LIN {X 0,Y 658.001,Z 1135.753,A -85,B 0,C 180,E1 30891.202,E2 30891.202} C_VEL
LIN {X 0,Y 657.305,Z 1150.031,A -85,B 0,C 180,E1 30888.997,E2 30888.997} C_VEL
LIN {X 0,Y 656.752,Z 1162.678,A -85,B 0,C 180,E1 30886.723,E2 30886.723} C_VEL
LIN {X 0,Y 656.451,Z 1171.896,A -85,B 0,C 180,E1 30884.826,E2 30884.826} C_VEL
LIN {X 0,Y 656.232,Z 1179.871,A -85,B 0,C 180,E1 30882.943,E2 30882.943} C_VEL
LIN {X 0,Y 656.05,Z 1187.892,A -85,B 0,C 180,E1 30880.716,E2 30880.716} C_VEL
LIN {X 0,Y 655.97,Z 1194.694,A -85,B 0,C 180,E1 30878.326,E2 30878.326} C_VEL
LIN {X 0,Y 655.929,Z 1199.41,A -85,B 0,C 180,E1 30876.125,E2 30876.125} C_VEL
LIN {X 0,Y 655.91,Z 1202.789,A -85,B 0,C 180,E1 30873.846,E2 30873.846} C_VEL
LIN {X 0,Y 655.911,Z 1204.624,A -85,B 0,C 180,E1 30871.485,E2 30871.485} C_VEL
LIN {X 0,Y 655.893,Z 1204.849,A -85,B 0,C 180,E1 30869.389,E2 30869.389} C_VEL
LIN {X 0,Y 655.908,Z 1203.947,A -85,B 0,C 180,E1 30867.379,E2 30867.379} C_VEL
LIN {X 0,Y 655.919,Z 1201.428,A -85,B 0,C 180,E1 30865.103,E2 30865.103} C_VEL
LIN {X 0,Y 655.949,Z 1197.152,A -85,B 0,C 180,E1 30862.732,E2 30862.732} C_VEL
LIN {X 0,Y 656.009,Z 1191.376,A -85,B 0,C 180,E1 30860.437,E2 30860.437} C_VEL
LIN {X 0,Y 656.126,Z 1184.279,A -85,B 0,C 180,E1 30858.217,E2 30858.217} C_VEL
LIN {X 0,Y 656.39,Z 1174.089,A -85,B 0,C 180,E1 30855.658,E2 30855.658} C_VEL
LIN {X 0,Y 656.694,Z 1164.274,A -85,B 0,C 180,E1 30853.587,E2 30853.587} C_VEL
LIN {X 0,Y 657.112,Z 1154.137,A -85,B 0,C 180,E1 30851.716,E2 30851.716} C_VEL
LIN {X 0,Y 657.764,Z 1140.78,A -85,B 0,C 180,E1 30849.536,E2 30849.536} C_VEL
LIN {X 0,Y 658.6,Z 1125.104,A -85,B 0,C 180,E1 30847.318,E2 30847.318} C_VEL
LIN {X 0,Y 659.475,Z 1110.399,A -85,B 0,C 180,E1 30845.467,E2 30845.467} C_VEL
LIN {X 0,Y 660.73,Z 1092.314,A -85,B 0,C 180,E1 30843.428,E2 30843.428} C_VEL
LIN {X 0,Y 662,Z 1073.819,A -85,B 0,C 180,E1 30841.591,E2 30841.591} C_VEL
LIN {X 0,Y 663.289,Z 1056.842,A -85,B 0,C 180,E1 30840.069,E2 30840.069} C_VEL
LIN {X 0,Y 664.962,Z 1035.53,A -85,B 0,C 180,E1 30838.348,E2 30838.348} C_VEL
LIN {X 0,Y 666.618,Z 1013.004,A -85,B 0,C 180,E1 30836.756,E2 30836.756} C_VEL
LIN {X 0,Y 668.131,Z 993.022,A -85,B 0,C 180,E1 30835.499,E2 30835.499} C_VEL
LIN {X 0,Y 669.972,Z 968.967,A -85,B 0,C 180,E1 30834.161,E2 30834.161} C_VEL
LIN {X 0,Y 671.656,Z 944.001,A -85,B 0,C 180,E1 30832.976,E2 30832.976} C_VEL
LIN {X 0,Y 672.975,Z 923.055,A -85,B 0,C 180,E1 30832.114,E2 30832.114} C_VEL
LIN {X 0,Y 674.098,Z 902.837,A -85,B 0,C 180,E1 30831.392,E2 30831.392} C_VEL
LIN {X 0,Y 675.312,Z 879.657,A -85,B 0,C 180,E1 30830.692,E2 30830.692} C_VEL
LIN {X 0,Y 676.519,Z 851.801,A -85,B 0,C 180,E1 30830.029,E2 30830.029} C_VEL
LIN {X 0,Y 677.299,Z 826.241,A -85,B 0,C 180,E1 30829.585,E2 30829.585} C_VEL
LIN {X 0,Y 680.373,Z 611.931,A -85,B 0,C 180,E1 30826.813,E2 30826.813} C_VEL
LIN {X 0,Y 683.542,Z 400.047,A -85,B 0,C 180,E1 30824.005,E2 30824.005} C_VEL
LIN {X 0,Y 683.78,Z 375.573,A -85,B 0,C 180,E1 30823.663,E2 30823.663} C_VEL
LIN {X 0,Y 678.293,Z 349.765,A -85,B 0,C 180,E1 30822.77,E2 30822.77} C_VEL
LIN {X 0,Y 678.555,Z 340.602,A -85,B 0,C 180,E1 30822.168,E2 30822.168} C_VEL
LIN {X 0,Y 667.4,Z 318.931,A -85,B 0,C 180,E1 30819.66,E2 30819.66} C_VEL
LIN {X 0,Y 660.624,Z 305.776,A -85,B 0,C 180,E1 30818.026,E2 30818.026} C_VEL
LIN {X 0,Y 658.168,Z 301.139,A -85,B 0,C 180,E1 30817.422,E2 30817.422} C_VEL
LIN {X 0,Y 656.727,Z 297.652,A -85,B 0,C 180,E1 30816.96,E2 30816.96} C_VEL
LIN {X 0,Y 656.684,Z 297.427,A -85,B 0,C 180,E1 30813.974,E2 30813.974} C_VEL
LIN {X 0,Y 656.694,Z 297.401,A -85,B 0,C 180,E1 30810.974,E2 30810.974} C_VEL
LIN {X 0,Y 656.692,Z 297.415,A -85,B 0,C 180,E1 30807.967,E2 30807.967} C_VEL
LIN {X 0,Y 656.698,Z 297.426,A -85,B 0,C 180,E1 30804.946,E2 30804.946} C_VEL
LIN {X 0,Y 656.696,Z 297.397,A -85,B 0,C 180,E1 30801.903,E2 30801.903} C_VEL
LIN {X 0,Y 656.699,Z 297.431,A -85,B 0,C 180,E1 30798.832,E2 30798.832} C_VEL
LIN {X 0,Y 656.694,Z 297.39,A -85,B 0,C 180,E1 30795.725,E2 30795.725} C_VEL
LIN {X 0,Y 656.695,Z 297.429,A -85,B 0,C 180,E1 30792.665,E2 30792.665} C_VEL
LIN {X 0,Y 656.696,Z 297.389,A -85,B 0,C 180,E1 30789.553,E2 30789.553} C_VEL
LIN {X 0,Y 656.689,Z 297.431,A -85,B 0,C 180,E1 30786.47,E2 30786.47} C_VEL
LIN {X 0,Y 656.702,Z 297.422,A -85,B 0,C 180,E1 30783.404,E2 30783.404} C_VEL
LIN {X 0,Y 656.686,Z 297.43,A -85,B 0,C 180,E1 30780.349,E2 30780.349} C_VEL
LIN {X 0,Y 656.703,Z 297.416,A -85,B 0,C 180,E1 30777.295,E2 30777.295} C_VEL
LIN {X 0,Y 656.686,Z 297.423,A -85,B 0,C 180,E1 30774.232,E2 30774.232} C_VEL
LIN {X 0,Y 656.707,Z 297.424,A -85,B 0,C 180,E1 30771.154,E2 30771.154} C_VEL
LIN {X 0,Y 656.682,Z 297.428,A -85,B 0,C 180,E1 30768.049,E2 30768.049} C_VEL
LIN {X 0,Y 656.71,Z 297.424,A -85,B 0,C 180,E1 30764.999,E2 30764.999} C_VEL
LIN {X 0,Y 656.678,Z 297.432,A -85,B 0,C 180,E1 30761.903,E2 30761.903} C_VEL
LIN {X 0,Y 656.709,Z 297.42,A -85,B 0,C 180,E1 30758.847,E2 30758.847} C_VEL
LIN {X 0,Y 656.67,Z 297.403,A -85,B 0,C 180,E1 30755.725,E2 30755.725} C_VEL
LIN {X 0,Y 656.705,Z 297.417,A -85,B 0,C 180,E1 30752.722,E2 30752.722} C_VEL
LIN {X 0,Y 656.67,Z 297.407,A -85,B 0,C 180,E1 30749.634,E2 30749.634} C_VEL
LIN {X 0,Y 656.698,Z 297.42,A -85,B 0,C 180,E1 30746.656,E2 30746.656} C_VEL
LIN {X 0,Y 656.666,Z 297.4,A -85,B 0,C 180,E1 30743.509,E2 30743.509} C_VEL
LIN {X 0,Y 656.695,Z 297.428,A -85,B 0,C 180,E1 30740.528,E2 30740.528} C_VEL
LIN {X 0,Y 656.698,Z 297.428,A -85,B 0,C 180,E1 30740.497,E2 30740.497} C_VEL
LIN {X 0,Y 655.768,Z 297.543,A -85,B 0,C 180,E1 30739.825,E2 30739.825} C_VEL
LIN {X 0,Y 649.201,Z 298.332,A -85,B 0,C 180,E1 30737.893,E2 30737.893} C_VEL
LIN {X 0,Y 648.731,Z 298.392,A -85,B 0,C 180,E1 30737.451,E2 30737.451} C_VEL
LIN {X 0,Y 648.729,Z 298.404,A -85,B 0,C 180,E1 30734.595,E2 30734.595} C_VEL
LIN {X 0,Y 648.737,Z 298.422,A -85,B 0,C 180,E1 30731.357,E2 30731.357} C_VEL
LIN {X 0,Y 648.807,Z 298.65,A -85,B 0,C 180,E1 30729.906,E2 30729.906} C_VEL
LIN {X 0,Y 650.17,Z 302.073,A -85,B 0,C 180,E1 30729.429,E2 30729.429} C_VEL
LIN {X 0,Y 656.974,Z 316.09,A -85,B 0,C 180,E1 30727.538,E2 30727.538} C_VEL
LIN {X 0,Y 663.735,Z 330.81,A -85,B 0,C 180,E1 30725.66,E2 30725.66} C_VEL
LIN {X 0,Y 667.446,Z 339.825,A -85,B 0,C 180,E1 30724.594,E2 30724.594} C_VEL
LIN {X 0,Y 667.126,Z 347.451,A -85,B 0,C 180,E1 30724.054,E2 30724.054} C_VEL
LIN {X 0,Y 673.211,Z 374.417,A -85,B 0,C 180,E1 30723.133,E2 30723.133} C_VEL
LIN {X 0,Y 669.499,Z 604.5,A -85,B 0,C 180,E1 30720.151,E2 30720.151} C_VEL
LIN {X 0,Y 667.067,Z 780.533,A -85,B 0,C 180,E1 30717.931,E2 30717.931} C_VEL
LIN {X 0,Y 666.246,Z 807.391,A -85,B 0,C 180,E1 30717.446,E2 30717.446} C_VEL
LIN {X 0,Y 665.258,Z 830.021,A -85,B 0,C 180,E1 30716.891,E2 30716.891} C_VEL
LIN {X 0,Y 664.302,Z 849.337,A -85,B 0,C 180,E1 30716.312,E2 30716.312} C_VEL
LIN {X 0,Y 663.135,Z 870.21,A -85,B 0,C 180,E1 30715.571,E2 30715.571} C_VEL
LIN {X 0,Y 661.528,Z 895.398,A -85,B 0,C 180,E1 30714.506,E2 30714.506} C_VEL
LIN {X 0,Y 660.09,Z 916.05,A -85,B 0,C 180,E1 30713.476,E2 30713.476} C_VEL
LIN {X 0,Y 658.632,Z 936.675,A -85,B 0,C 180,E1 30712.304,E2 30712.304} C_VEL
LIN {X 0,Y 656.942,Z 959.384,A -85,B 0,C 180,E1 30710.817,E2 30710.817} C_VEL
LIN {X 0,Y 655.495,Z 978.127,A -85,B 0,C 180,E1 30709.422,E2 30709.422} C_VEL
LIN {X 0,Y 654.046,Z 998.172,A -85,B 0,C 180,E1 30707.743,E2 30707.743} C_VEL
LIN {X 0,Y 652.711,Z 1016.296,A -85,B 0,C 180,E1 30706.006,E2 30706.006} C_VEL
LIN {X 0,Y 651.571,Z 1033.024,A -85,B 0,C 180,E1 30704.213,E2 30704.213} C_VEL
LIN {X 0,Y 650.501,Z 1049.809,A -85,B 0,C 180,E1 30702.156,E2 30702.156} C_VEL
LIN {X 0,Y 649.761,Z 1063.29,A -85,B 0,C 180,E1 30700.282,E2 30700.282} C_VEL
LIN {X 0,Y 649.074,Z 1077.256,A -85,B 0,C 180,E1 30698.058,E2 30698.058} C_VEL
LIN {X 0,Y 648.632,Z 1087.822,A -85,B 0,C 180,E1 30696.106,E2 30696.106} C_VEL
LIN {X 0,Y 648.338,Z 1097.37,A -85,B 0,C 180,E1 30694.068,E2 30694.068} C_VEL
LIN {X 0,Y 648.105,Z 1106.283,A -85,B 0,C 180,E1 30691.768,E2 30691.768} C_VEL
LIN {X 0,Y 647.99,Z 1112.419,A -85,B 0,C 180,E1 30689.823,E2 30689.823} C_VEL
LIN {X 0,Y 647.948,Z 1117.134,A -85,B 0,C 180,E1 30687.966,E2 30687.966} C_VEL
LIN {X 0,Y 647.907,Z 1121.473,A -85,B 0,C 180,E1 30685.663,E2 30685.663} C_VEL
LIN {X 0,Y 647.912,Z 1123.863,A -85,B 0,C 180,E1 30683.532,E2 30683.532} C_VEL
LIN {X 0,Y 647.91,Z 1124.829,A -85,B 0,C 180,E1 30681.659,E2 30681.659} C_VEL
LIN {X 0,Y 647.904,Z 1124.662,A -85,B 0,C 180,E1 30679.598,E2 30679.598} C_VEL
LIN {X 0,Y 647.916,Z 1122.754,A -85,B 0,C 180,E1 30677.248,E2 30677.248} C_VEL
LIN {X 0,Y 647.915,Z 1119.922,A -85,B 0,C 180,E1 30675.34,E2 30675.34} C_VEL
LIN {X 0,Y 647.959,Z 1116.115,A -85,B 0,C 180,E1 30673.505,E2 30673.505} C_VEL
LIN {X 0,Y 648.043,Z 1110.121,A -85,B 0,C 180,E1 30671.281,E2 30671.281} C_VEL
LIN {X 0,Y 648.202,Z 1102.181,A -85,B 0,C 180,E1 30669.031,E2 30669.031} C_VEL
LIN {X 0,Y 648.411,Z 1094.625,A -85,B 0,C 180,E1 30667.229,E2 30667.229} C_VEL
LIN {X 0,Y 648.775,Z 1084.74,A -85,B 0,C 180,E1 30665.199,E2 30665.199} C_VEL
LIN {X 0,Y 649.31,Z 1072.034,A -85,B 0,C 180,E1 30662.982,E2 30662.982} C_VEL
LIN {X 0,Y 649.949,Z 1059.761,A -85,B 0,C 180,E1 30661.115,E2 30661.115} C_VEL
LIN {X 0,Y 650.876,Z 1043.982,A -85,B 0,C 180,E1 30659.006,E2 30659.006} C_VEL
LIN {X 0,Y 651.867,Z 1028.543,A -85,B 0,C 180,E1 30657.201,E2 30657.201} C_VEL
LIN {X 0,Y 653.028,Z 1011.944,A -85,B 0,C 180,E1 30655.464,E2 30655.464} C_VEL
LIN {X 0,Y 654.458,Z 992.162,A -85,B 0,C 180,E1 30653.646,E2 30653.646} C_VEL
LIN {X 0,Y 655.805,Z 974.433,A -85,B 0,C 180,E1 30652.201,E2 30652.201} C_VEL
LIN {X 0,Y 657.481,Z 952.02,A -85,B 0,C 180,E1 30650.585,E2 30650.585} C_VEL
LIN {X 0,Y 658.943,Z 932.021,A -85,B 0,C 180,E1 30649.33,E2 30649.33} C_VEL
LIN {X 0,Y 660.527,Z 910.49,A -85,B 0,C 180,E1 30648.14,E2 30648.14} C_VEL
LIN {X 0,Y 662.114,Z 886.692,A -85,B 0,C 180,E1 30647.015,E2 30647.015} C_VEL
LIN {X 0,Y 663.382,Z 865.65,A -85,B 0,C 180,E1 30646.167,E2 30646.167} C_VEL
LIN {X 0,Y 664.58,Z 844.003,A -85,B 0,C 180,E1 30645.425,E2 30645.425} C_VEL
LIN {X 0,Y 665.807,Z 817,A -85,B 0,C 180,E1 30644.682,E2 30644.682} C_VEL
LIN {X 0,Y 666.623,Z 794.883,A -85,B 0,C 180,E1 30644.217,E2 30644.217} C_VEL
LIN {X 0,Y 667.316,Z 769.851,A -85,B 0,C 180,E1 30643.828,E2 30643.828} C_VEL
LIN {X 0,Y 670.628,Z 527.96,A -85,B 0,C 180,E1 30640.783,E2 30640.783} C_VEL
LIN {X 0,Y 673.17,Z 373.299,A -85,B 0,C 180,E1 30638.744,E2 30638.744} C_VEL
LIN {X 0,Y 667.143,Z 346.712,A -85,B 0,C 180,E1 30637.807,E2 30637.807} C_VEL
LIN {X 0,Y 667.583,Z 340.05,A -85,B 0,C 180,E1 30637.317,E2 30637.317} C_VEL
LIN {X 0,Y 661.902,Z 326.465,A -85,B 0,C 180,E1 30635.669,E2 30635.669} C_VEL
LIN {X 0,Y 654.624,Z 310.93,A -85,B 0,C 180,E1 30633.568,E2 30633.568} C_VEL
LIN {X 0,Y 652.075,Z 305.952,A -85,B 0,C 180,E1 30632.831,E2 30632.831} C_VEL
LIN {X 0,Y 650.535,Z 302.539,A -85,B 0,C 180,E1 30632.336,E2 30632.336} C_VEL
LIN {X 0,Y 648.827,Z 298.862,A -85,B 0,C 180,E1 30631.767,E2 30631.767} C_VEL
LIN {X 0,Y 648.76,Z 298.417,A -85,B 0,C 180,E1 30631.201,E2 30631.201} C_VEL
LIN {X 0,Y 648.766,Z 298.416,A -85,B 0,C 180,E1 30628.039,E2 30628.039} C_VEL
LIN {X 0,Y 648.748,Z 298.402,A -85,B 0,C 180,E1 30624.883,E2 30624.883} C_VEL
LIN {X 0,Y 648.757,Z 298.39,A -85,B 0,C 180,E1 30621.805,E2 30621.805} C_VEL
LIN {X 0,Y 648.752,Z 298.418,A -85,B 0,C 180,E1 30618.698,E2 30618.698} C_VEL
LIN {X 0,Y 648.756,Z 298.407,A -85,B 0,C 180,E1 30615.582,E2 30615.582} C_VEL
LIN {X 0,Y 648.751,Z 298.392,A -85,B 0,C 180,E1 30612.552,E2 30612.552} C_VEL
LIN {X 0,Y 648.757,Z 298.42,A -85,B 0,C 180,E1 30609.474,E2 30609.474} C_VEL
LIN {X 0,Y 648.751,Z 298.388,A -85,B 0,C 180,E1 30606.371,E2 30606.371} C_VEL
LIN {X 0,Y 648.753,Z 298.409,A -85,B 0,C 180,E1 30603.269,E2 30603.269} C_VEL
LIN {X 0,Y 648.753,Z 298.403,A -85,B 0,C 180,E1 30600.177,E2 30600.177} C_VEL
LIN {X 0,Y 648.75,Z 298.395,A -85,B 0,C 180,E1 30597.085,E2 30597.085} C_VEL
LIN {X 0,Y 648.753,Z 298.412,A -85,B 0,C 180,E1 30593.984,E2 30593.984} C_VEL
LIN {X 0,Y 648.747,Z 298.387,A -85,B 0,C 180,E1 30590.955,E2 30590.955} C_VEL
LIN {X 0,Y 648.758,Z 298.416,A -85,B 0,C 180,E1 30587.901,E2 30587.901} C_VEL
LIN {X 0,Y 648.747,Z 298.393,A -85,B 0,C 180,E1 30584.81,E2 30584.81} C_VEL
LIN {X 0,Y 648.761,Z 298.412,A -85,B 0,C 180,E1 30581.768,E2 30581.768} C_VEL
LIN {X 0,Y 648.749,Z 298.414,A -85,B 0,C 180,E1 30578.67,E2 30578.67} C_VEL
LIN {X 0,Y 648.76,Z 298.387,A -85,B 0,C 180,E1 30575.603,E2 30575.603} C_VEL
LIN {X 0,Y 648.75,Z 298.408,A -85,B 0,C 180,E1 30572.559,E2 30572.559} C_VEL
LIN {X 0,Y 648.764,Z 298.417,A -85,B 0,C 180,E1 30569.429,E2 30569.429} C_VEL
LIN {X 0,Y 648.746,Z 298.416,A -85,B 0,C 180,E1 30566.331,E2 30566.331} C_VEL
LIN {X 0,Y 648.783,Z 298.677,A -85,B 0,C 180,E1 30563.835,E2 30563.835} C_VEL
LIN {X 0,Y 650.131,Z 301.988,A -85,B 0,C 180,E1 30563.363,E2 30563.363} C_VEL
LIN {X 0,Y 651.245,Z 303.643,A -85,B 0,C 180,E1 30563.107,E2 30563.107} C_VEL
LIN {X 0,Y 658.408,Z 317.778,A -85,B 0,C 180,E1 30561.267,E2 30561.267} C_VEL
LIN {X 0,Y 671.527,Z 343.462,A -85,B 0,C 180,E1 30558.241,E2 30558.241} C_VEL
LIN {X 0,Y 672.392,Z 345.474,A -85,B 0,C 180,E1 30558.031,E2 30558.031} C_VEL
LIN {X 0,Y 672.364,Z 350.69,A -85,B 0,C 180,E1 30557.728,E2 30557.728} C_VEL
LIN {X 0,Y 678.337,Z 378.966,A -85,B 0,C 180,E1 30556.77,E2 30556.77} C_VEL
LIN {X 0,Y 674.876,Z 590.194,A -85,B 0,C 180,E1 30553.941,E2 30553.941} C_VEL
LIN {X 0,Y 671.51,Z 814.244,A -85,B 0,C 180,E1 30551.028,E2 30551.028} C_VEL
LIN {X 0,Y 670.692,Z 842.215,A -85,B 0,C 180,E1 30550.596,E2 30550.596} C_VEL
LIN {X 0,Y 669.734,Z 865.671,A -85,B 0,C 180,E1 30550.102,E2 30550.102} C_VEL
LIN {X 0,Y 668.493,Z 890.858,A -85,B 0,C 180,E1 30549.428,E2 30549.428} C_VEL
LIN {X 0,Y 666.809,Z 918.654,A -85,B 0,C 180,E1 30548.487,E2 30548.487} C_VEL
LIN {X 0,Y 665.363,Z 939.924,A -85,B 0,C 180,E1 30547.63,E2 30547.63} C_VEL
LIN {X 0,Y 663.854,Z 960.721,A -85,B 0,C 180,E1 30546.669,E2 30546.669} C_VEL
LIN {X 0,Y 662.097,Z 983.908,A -85,B 0,C 180,E1 30545.443,E2 30545.443} C_VEL
LIN {X 0,Y 660.055,Z 1008.604,A -85,B 0,C 180,E1 30543.932,E2 30543.932} C_VEL
LIN {X 0,Y 658.449,Z 1027.581,A -85,B 0,C 180,E1 30542.62,E2 30542.62} C_VEL
LIN {X 0,Y 656.823,Z 1047.086,A -85,B 0,C 180,E1 30541.118,E2 30541.118} C_VEL
LIN {X 0,Y 654.983,Z 1069.757,A -85,B 0,C 180,E1 30539.141,E2 30539.141} C_VEL
LIN {X 0,Y 653.645,Z 1086.388,A -85,B 0,C 180,E1 30537.514,E2 30537.514} C_VEL
LIN {X 0,Y 652.369,Z 1103.305,A -85,B 0,C 180,E1 30535.679,E2 30535.679} C_VEL
LIN {X 0,Y 651.104,Z 1121.565,A -85,B 0,C 180,E1 30533.436,E2 30533.436} C_VEL
LIN {X 0,Y 650.245,Z 1135.429,A -85,B 0,C 180,E1 30531.515,E2 30531.515} C_VEL
LIN {X 0,Y 649.487,Z 1149.549,A -85,B 0,C 180,E1 30529.313,E2 30529.313} C_VEL
LIN {X 0,Y 648.874,Z 1162.214,A -85,B 0,C 180,E1 30527.024,E2 30527.024} C_VEL
LIN {X 0,Y 648.513,Z 1171.487,A -85,B 0,C 180,E1 30525.103,E2 30525.103} C_VEL
LIN {X 0,Y 648.28,Z 1179.515,A -85,B 0,C 180,E1 30523.195,E2 30523.195} C_VEL
LIN {X 0,Y 648.084,Z 1187.034,A -85,B 0,C 180,E1 30521.112,E2 30521.112} C_VEL
LIN {X 0,Y 647.987,Z 1193.816,A -85,B 0,C 180,E1 30518.787,E2 30518.787} C_VEL
LIN {X 0,Y 647.935,Z 1199.101,A -85,B 0,C 180,E1 30516.372,E2 30516.372} C_VEL
LIN {X 0,Y 647.918,Z 1202.476,A -85,B 0,C 180,E1 30514.159,E2 30514.159} C_VEL
LIN {X 0,Y 647.908,Z 1204.549,A -85,B 0,C 180,E1 30511.769,E2 30511.769} C_VEL
LIN {X 0,Y 647.892,Z 1204.872,A -85,B 0,C 180,E1 30509.47,E2 30509.47} C_VEL
LIN {X 0,Y 647.909,Z 1203.944,A -85,B 0,C 180,E1 30507.347,E2 30507.347} C_VEL
LIN {X 0,Y 647.922,Z 1201.428,A -85,B 0,C 180,E1 30505.043,E2 30505.043} C_VEL
LIN {X 0,Y 647.951,Z 1197.152,A -85,B 0,C 180,E1 30502.642,E2 30502.642} C_VEL
LIN {X 0,Y 648.018,Z 1191.373,A -85,B 0,C 180,E1 30500.318,E2 30500.318} C_VEL
LIN {X 0,Y 648.146,Z 1184.279,A -85,B 0,C 180,E1 30498.07,E2 30498.07} C_VEL
LIN {X 0,Y 648.439,Z 1174.338,A -85,B 0,C 180,E1 30495.535,E2 30495.535} C_VEL
LIN {X 0,Y 648.771,Z 1164.544,A -85,B 0,C 180,E1 30493.434,E2 30493.434} C_VEL
LIN {X 0,Y 649.238,Z 1154.237,A -85,B 0,C 180,E1 30491.503,E2 30491.503} C_VEL
LIN {X 0,Y 649.924,Z 1141.364,A -85,B 0,C 180,E1 30489.372,E2 30489.372} C_VEL
LIN {X 0,Y 650.838,Z 1125.803,A -85,B 0,C 180,E1 30487.128,E2 30487.128} C_VEL
LIN {X 0,Y 651.804,Z 1111.152,A -85,B 0,C 180,E1 30485.252,E2 30485.252} C_VEL
LIN {X 0,Y 653.113,Z 1093.727,A -85,B 0,C 180,E1 30483.251,E2 30483.251} C_VEL
LIN {X 0,Y 654.547,Z 1074.832,A -85,B 0,C 180,E1 30481.337,E2 30481.337} C_VEL
LIN {X 0,Y 655.937,Z 1057.951,A -85,B 0,C 180,E1 30479.8,E2 30479.8} C_VEL
LIN {X 0,Y 657.511,Z 1039.194,A -85,B 0,C 180,E1 30478.254,E2 30478.254} C_VEL
LIN {X 0,Y 659.487,Z 1015.132,A -85,B 0,C 180,E1 30476.501,E2 30476.501} C_VEL
LIN {X 0,Y 661.142,Z 994.951,A -85,B 0,C 180,E1 30475.207,E2 30475.207} C_VEL
LIN {X 0,Y 662.831,Z 974.061,A -85,B 0,C 180,E1 30474.017,E2 30474.017} C_VEL
LIN {X 0,Y 664.822,Z 948.476,A -85,B 0,C 180,E1 30472.747,E2 30472.747} C_VEL
LIN {X 0,Y 666.407,Z 925.174,A -85,B 0,C 180,E1 30471.764,E2 30471.764} C_VEL
LIN {X 0,Y 667.661,Z 904.465,A -85,B 0,C 180,E1 30471.01,E2 30471.01} C_VEL
LIN {X 0,Y 668.911,Z 882.309,A -85,B 0,C 180,E1 30470.327,E2 30470.327} C_VEL
LIN {X 0,Y 670.161,Z 856.683,A -85,B 0,C 180,E1 30469.689,E2 30469.689} C_VEL
LIN {X 0,Y 671.132,Z 829.115,A -85,B 0,C 180,E1 30469.183,E2 30469.183} C_VEL
LIN {X 0,Y 672.99,Z 712.974,A -85,B 0,C 180,E1 30467.665,E2 30467.665} C_VEL
LIN {X 0,Y 676.471,Z 490.787,A -85,B 0,C 180,E1 30464.739,E2 30464.739} C_VEL
LIN {X 0,Y 678.217,Z 377.64,A -85,B 0,C 180,E1 30463.199,E2 30463.199} C_VEL
LIN {X 0,Y 672.239,Z 349.327,A -85,B 0,C 180,E1 30462.209,E2 30462.209} C_VEL
LIN {X 0,Y 672.405,Z 345.187,A -85,B 0,C 180,E1 30461.946,E2 30461.946} C_VEL
LIN {X 0,Y 661.741,Z 324.301,A -85,B 0,C 180,E1 30459.504,E2 30459.504} C_VEL
LIN {X 0,Y 655.01,Z 311.17,A -85,B 0,C 180,E1 30457.855,E2 30457.855} C_VEL
LIN {X 0,Y 650.486,Z 302.474,A -85,B 0,C 180,E1 30456.723,E2 30456.723} C_VEL
LIN {X 0,Y 648.805,Z 298.775,A -85,B 0,C 180,E1 30456.228,E2 30456.228} C_VEL
LIN {X 0,Y 648.766,Z 298.42,A -85,B 0,C 180,E1 30455.385,E2 30455.385} C_VEL
LIN {X 0,Y 648.756,Z 298.391,A -85,B 0,C 180,E1 30452.209,E2 30452.209} C_VEL
LIN {X 0,Y 648.764,Z 298.421,A -85,B 0,C 180,E1 30449.092,E2 30449.092} C_VEL
LIN {X 0,Y 648.752,Z 298.395,A -85,B 0,C 180,E1 30445.958,E2 30445.958} C_VEL
LIN {X 0,Y 648.755,Z 298.398,A -85,B 0,C 180,E1 30442.855,E2 30442.855} C_VEL
LIN {X 0,Y 648.758,Z 298.409,A -85,B 0,C 180,E1 30439.82,E2 30439.82} C_VEL
LIN {X 0,Y 648.753,Z 298.385,A -85,B 0,C 180,E1 30436.751,E2 30436.751} C_VEL
LIN {X 0,Y 648.759,Z 298.409,A -85,B 0,C 180,E1 30433.639,E2 30433.639} C_VEL
LIN {X 0,Y 648.749,Z 298.386,A -85,B 0,C 180,E1 30430.568,E2 30430.568} C_VEL
LIN {X 0,Y 648.758,Z 298.406,A -85,B 0,C 180,E1 30427.439,E2 30427.439} C_VEL
LIN {X 0,Y 648.747,Z 298.413,A -85,B 0,C 180,E1 30424.331,E2 30424.331} C_VEL
LIN {X 0,Y 648.76,Z 298.411,A -85,B 0,C 180,E1 30421.236,E2 30421.236} C_VEL
LIN {X 0,Y 648.745,Z 298.411,A -85,B 0,C 180,E1 30418.234,E2 30418.234} C_VEL
LIN {X 0,Y 648.763,Z 298.415,A -85,B 0,C 180,E1 30415.137,E2 30415.137} C_VEL
LIN {X 0,Y 648.742,Z 298.42,A -85,B 0,C 180,E1 30412.116,E2 30412.116} C_VEL
LIN {X 0,Y 648.766,Z 298.412,A -85,B 0,C 180,E1 30409.029,E2 30409.029} C_VEL
LIN {X 0,Y 648.737,Z 298.42,A -85,B 0,C 180,E1 30405.905,E2 30405.905} C_VEL
LIN {X 0,Y 648.767,Z 298.405,A -85,B 0,C 180,E1 30402.847,E2 30402.847} C_VEL
LIN {X 0,Y 648.735,Z 298.413,A -85,B 0,C 180,E1 30399.803,E2 30399.803} C_VEL
LIN {X 0,Y 648.77,Z 298.412,A -85,B 0,C 180,E1 30396.762,E2 30396.762} C_VEL
LIN {X 0,Y 648.73,Z 298.396,A -85,B 0,C 180,E1 30393.647,E2 30393.647} C_VEL
LIN {X 0,Y 648.771,Z 298.413,A -85,B 0,C 180,E1 30390.652,E2 30390.652} C_VEL
LIN {X 0,Y 648.729,Z 298.397,A -85,B 0,C 180,E1 30387.563,E2 30387.563} C_VEL
LIN {X 0,Y 648.76,Z 298.412,A -85,B 0,C 180,E1 30384.584,E2 30384.584} C_VEL
LIN {X 0,Y 648.73,Z 298.408,A -85,B 0,C 180,E1 30381.487,E2 30381.487} C_VEL
LIN {X 0,Y 648.736,Z 298.394,A -85,B 0,C 180,E1 30378.607,E2 30378.607} C_VEL
LIN {X 0,Y 648.731,Z 298.392,A -85,B 0,C 180,E1 30377.451,E2 30377.451} C_VEL
LIN {X 0,Y 647.701,Z 298.534,A -85,B 0,C 180,E1 30376.771,E2 30376.771} C_VEL
LIN {X 0,Y 641.297,Z 299.335,A -85,B 0,C 180,E1 30374.863,E2 30374.863} C_VEL
LIN {X 0,Y 640.811,Z 299.381,A -85,B 0,C 180,E1 30374.367,E2 30374.367} C_VEL
LIN {X 0,Y 640.785,Z 299.41,A -85,B 0,C 180,E1 30371.183,E2 30371.183} C_VEL
LIN {X 0,Y 640.85,Z 299.859,A -85,B 0,C 180,E1 30370.623,E2 30370.623} C_VEL
LIN {X 0,Y 642.496,Z 303.399,A -85,B 0,C 180,E1 30370.111,E2 30370.111} C_VEL
LIN {X 0,Y 651.081,Z 321.278,A -85,B 0,C 180,E1 30367.677,E2 30367.677} C_VEL
LIN {X 0,Y 658.123,Z 336.818,A -85,B 0,C 180,E1 30365.69,E2 30365.69} C_VEL
LIN {X 0,Y 661.013,Z 344.169,A -85,B 0,C 180,E1 30364.821,E2 30364.821} C_VEL
LIN {X 0,Y 660.993,Z 347.691,A -85,B 0,C 180,E1 30364.591,E2 30364.591} C_VEL
LIN {X 0,Y 667.477,Z 375.98,A -85,B 0,C 180,E1 30363.596,E2 30363.596} C_VEL
LIN {X 0,Y 663.188,Z 617.192,A -85,B 0,C 180,E1 30360.436,E2 30360.436} C_VEL
LIN {X 0,Y 660.659,Z 781.011,A -85,B 0,C 180,E1 30358.342,E2 30358.342} C_VEL
LIN {X 0,Y 659.755,Z 808.065,A -85,B 0,C 180,E1 30357.846,E2 30357.846} C_VEL
LIN {X 0,Y 658.735,Z 829.983,A -85,B 0,C 180,E1 30357.305,E2 30357.305} C_VEL
LIN {X 0,Y 657.735,Z 848.713,A -85,B 0,C 180,E1 30356.741,E2 30356.741} C_VEL
LIN {X 0,Y 656.51,Z 869.14,A -85,B 0,C 180,E1 30356.016,E2 30356.016} C_VEL
LIN {X 0,Y 654.859,Z 893.914,A -85,B 0,C 180,E1 30354.971,E2 30354.971} C_VEL
LIN {X 0,Y 653.207,Z 915.693,A -85,B 0,C 180,E1 30353.883,E2 30353.883} C_VEL
LIN {X 0,Y 651.612,Z 936.375,A -85,B 0,C 180,E1 30352.7,E2 30352.7} C_VEL
LIN {X 0,Y 649.744,Z 959.672,A -85,B 0,C 180,E1 30351.16,E2 30351.16} C_VEL
LIN {X 0,Y 648.239,Z 977.831,A -85,B 0,C 180,E1 30349.795,E2 30349.795} C_VEL
LIN {X 0,Y 646.648,Z 997.841,A -85,B 0,C 180,E1 30348.107,E2 30348.107} C_VEL
LIN {X 0,Y 645.232,Z 1015.685,A -85,B 0,C 180,E1 30346.381,E2 30346.381} C_VEL
LIN {X 0,Y 644.052,Z 1031.178,A -85,B 0,C 180,E1 30344.713,E2 30344.713} C_VEL
LIN {X 0,Y 642.857,Z 1048.656,A -85,B 0,C 180,E1 30342.577,E2 30342.577} C_VEL
LIN {X 0,Y 642.03,Z 1061.637,A -85,B 0,C 180,E1 30340.771,E2 30340.771} C_VEL
LIN {X 0,Y 641.294,Z 1075.389,A -85,B 0,C 180,E1 30338.608,E2 30338.608} C_VEL
LIN {X 0,Y 640.741,Z 1087.056,A -85,B 0,C 180,E1 30336.451,E2 30336.451} C_VEL
LIN {X 0,Y 640.432,Z 1095.898,A -85,B 0,C 180,E1 30334.567,E2 30334.567} C_VEL
LIN {X 0,Y 640.162,Z 1105.167,A -85,B 0,C 180,E1 30332.238,E2 30332.238} C_VEL
LIN {X 0,Y 640.022,Z 1111.983,A -85,B 0,C 180,E1 30330.089,E2 30330.089} C_VEL
LIN {X 0,Y 639.951,Z 1116.779,A -85,B 0,C 180,E1 30328.209,E2 30328.209} C_VEL
LIN {X 0,Y 639.92,Z 1120.797,A -85,B 0,C 180,E1 30326.148,E2 30326.148} C_VEL
LIN {X 0,Y 639.917,Z 1123.743,A -85,B 0,C 180,E1 30323.721,E2 30323.721} C_VEL
LIN {X 0,Y 639.914,Z 1124.812,A -85,B 0,C 180,E1 30321.735,E2 30321.735} C_VEL
LIN {X 0,Y 639.907,Z 1124.702,A -85,B 0,C 180,E1 30319.739,E2 30319.739} C_VEL
LIN {X 0,Y 639.916,Z 1122.959,A -85,B 0,C 180,E1 30317.364,E2 30317.364} C_VEL
LIN {X 0,Y 639.916,Z 1120.043,A -85,B 0,C 180,E1 30315.338,E2 30315.338} C_VEL
LIN {X 0,Y 639.963,Z 1116.272,A -85,B 0,C 180,E1 30313.48,E2 30313.48} C_VEL
LIN {X 0,Y 640.045,Z 1110.846,A -85,B 0,C 180,E1 30311.417,E2 30311.417} C_VEL
LIN {X 0,Y 640.219,Z 1102.817,A -85,B 0,C 180,E1 30309.045,E2 30309.045} C_VEL
LIN {X 0,Y 640.463,Z 1094.775,A -85,B 0,C 180,E1 30307.089,E2 30307.089} C_VEL
LIN {X 0,Y 640.863,Z 1084.872,A -85,B 0,C 180,E1 30305.025,E2 30305.025} C_VEL
LIN {X 0,Y 641.436,Z 1072.461,A -85,B 0,C 180,E1 30302.824,E2 30302.824} C_VEL
LIN {X 0,Y 642.126,Z 1060.239,A -85,B 0,C 180,E1 30300.934,E2 30300.934} C_VEL
LIN {X 0,Y 643.123,Z 1044.735,A -85,B 0,C 180,E1 30298.821,E2 30298.821} C_VEL
LIN {X 0,Y 644.233,Z 1028.891,A -85,B 0,C 180,E1 30296.942,E2 30296.942} C_VEL
LIN {X 0,Y 645.437,Z 1012.91,A -85,B 0,C 180,E1 30295.245,E2 30295.245} C_VEL
LIN {X 0,Y 647.014,Z 992.997,A -85,B 0,C 180,E1 30293.38,E2 30293.38} C_VEL
LIN {X 0,Y 648.46,Z 975.352,A -85,B 0,C 180,E1 30291.92,E2 30291.92} C_VEL
LIN {X 0,Y 650.16,Z 954.76,A -85,B 0,C 180,E1 30290.399,E2 30290.399} C_VEL
LIN {X 0,Y 651.88,Z 932.793,A -85,B 0,C 180,E1 30288.996,E2 30288.996} C_VEL
LIN {X 0,Y 653.469,Z 912.555,A -85,B 0,C 180,E1 30287.86,E2 30287.86} C_VEL
LIN {X 0,Y 655.265,Z 888.088,A -85,B 0,C 180,E1 30286.676,E2 30286.676} C_VEL
LIN {X 0,Y 656.674,Z 866.27,A -85,B 0,C 180,E1 30285.785,E2 30285.785} C_VEL
LIN {X 0,Y 657.908,Z 845.606,A -85,B 0,C 180,E1 30285.067,E2 30285.067} C_VEL
LIN {X 0,Y 659.214,Z 819.663,A -85,B 0,C 180,E1 30284.33,E2 30284.33} C_VEL
LIN {X 0,Y 660.153,Z 796.076,A -85,B 0,C 180,E1 30283.821,E2 30283.821} C_VEL
LIN {X 0,Y 660.846,Z 773.202,A -85,B 0,C 180,E1 30283.456,E2 30283.456} C_VEL
LIN {X 0,Y 664.232,Z 559.142,A -85,B 0,C 180,E1 30280.717,E2 30280.717} C_VEL
LIN {X 0,Y 667.522,Z 375.522,A -85,B 0,C 180,E1 30278.29,E2 30278.29} C_VEL
LIN {X 0,Y 661.013,Z 346.838,A -85,B 0,C 180,E1 30277.261,E2 30277.261} C_VEL
LIN {X 0,Y 661.046,Z 343.664,A -85,B 0,C 180,E1 30277.014,E2 30277.014} C_VEL
LIN {X 0,Y 655.108,Z 329.596,A -85,B 0,C 180,E1 30275.26,E2 30275.26} C_VEL
LIN {X 0,Y 648.439,Z 315.444,A -85,B 0,C 180,E1 30273.295,E2 30273.295} C_VEL
LIN {X 0,Y 644.599,Z 307.618,A -85,B 0,C 180,E1 30272.122,E2 30272.122} C_VEL
LIN {X 0,Y 642.368,Z 303.221,A -85,B 0,C 180,E1 30271.43,E2 30271.43} C_VEL
LIN {X 0,Y 640.832,Z 299.598,A -85,B 0,C 180,E1 30270.823,E2 30270.823} C_VEL
LIN {X 0,Y 640.822,Z 299.409,A -85,B 0,C 180,E1 30267.911,E2 30267.911} C_VEL
LIN {X 0,Y 640.808,Z 299.39,A -85,B 0,C 180,E1 30264.818,E2 30264.818} C_VEL
LIN {X 0,Y 640.818,Z 299.376,A -85,B 0,C 180,E1 30261.8,E2 30261.8} C_VEL
LIN {X 0,Y 640.812,Z 299.405,A -85,B 0,C 180,E1 30258.655,E2 30258.655} C_VEL
LIN {X 0,Y 640.817,Z 299.395,A -85,B 0,C 180,E1 30255.568,E2 30255.568} C_VEL
LIN {X 0,Y 640.811,Z 299.378,A -85,B 0,C 180,E1 30252.526,E2 30252.526} C_VEL
LIN {X 0,Y 640.818,Z 299.408,A -85,B 0,C 180,E1 30249.43,E2 30249.43} C_VEL
LIN {X 0,Y 640.811,Z 299.375,A -85,B 0,C 180,E1 30246.326,E2 30246.326} C_VEL
LIN {X 0,Y 640.816,Z 299.398,A -85,B 0,C 180,E1 30243.31,E2 30243.31} C_VEL
LIN {X 0,Y 640.815,Z 299.391,A -85,B 0,C 180,E1 30240.179,E2 30240.179} C_VEL
LIN {X 0,Y 640.813,Z 299.383,A -85,B 0,C 180,E1 30237.138,E2 30237.138} C_VEL
LIN {X 0,Y 640.815,Z 299.401,A -85,B 0,C 180,E1 30233.999,E2 30233.999} C_VEL
LIN {X 0,Y 640.807,Z 299.374,A -85,B 0,C 180,E1 30230.933,E2 30230.933} C_VEL
LIN {X 0,Y 640.819,Z 299.406,A -85,B 0,C 180,E1 30227.84,E2 30227.84} C_VEL
LIN {X 0,Y 640.808,Z 299.38,A -85,B 0,C 180,E1 30224.803,E2 30224.803} C_VEL
LIN {X 0,Y 640.82,Z 299.397,A -85,B 0,C 180,E1 30221.722,E2 30221.722} C_VEL
LIN {X 0,Y 640.81,Z 299.401,A -85,B 0,C 180,E1 30218.67,E2 30218.67} C_VEL
LIN {X 0,Y 640.82,Z 299.374,A -85,B 0,C 180,E1 30215.576,E2 30215.576} C_VEL
LIN {X 0,Y 640.807,Z 299.396,A -85,B 0,C 180,E1 30212.492,E2 30212.492} C_VEL
LIN {X 0,Y 640.825,Z 299.407,A -85,B 0,C 180,E1 30209.425,E2 30209.425} C_VEL
LIN {X 0,Y 640.808,Z 299.404,A -85,B 0,C 180,E1 30206.363,E2 30206.363} C_VEL
LIN {X 0,Y 640.862,Z 299.644,A -85,B 0,C 180,E1 30204.71,E2 30204.71} C_VEL
LIN {X 0,Y 642.331,Z 303.202,A -85,B 0,C 180,E1 30204.175,E2 30204.175} C_VEL
LIN {X 0,Y 643.431,Z 304.829,A -85,B 0,C 180,E1 30203.906,E2 30203.906} C_VEL
LIN {X 0,Y 650.383,Z 318.269,A -85,B 0,C 180,E1 30202.051,E2 30202.051} C_VEL
LIN {X 0,Y 663.784,Z 344.828,A -85,B 0,C 180,E1 30198.831,E2 30198.831} C_VEL
LIN {X 0,Y 666.095,Z 349.856,A -85,B 0,C 180,E1 30198.289,E2 30198.289} C_VEL
LIN {X 0,Y 672.814,Z 381.112,A -85,B 0,C 180,E1 30197.239,E2 30197.239} C_VEL
LIN {X 0,Y 669.07,Z 592.736,A -85,B 0,C 180,E1 30194.385,E2 30194.385} C_VEL
LIN {X 0,Y 665.418,Z 816.888,A -85,B 0,C 180,E1 30191.446,E2 30191.446} C_VEL
LIN {X 0,Y 664.559,Z 843.164,A -85,B 0,C 180,E1 30191.03,E2 30191.03} C_VEL
LIN {X 0,Y 663.55,Z 866.171,A -85,B 0,C 180,E1 30190.539,E2 30190.539} C_VEL
LIN {X 0,Y 662.21,Z 891.479,A -85,B 0,C 180,E1 30189.855,E2 30189.855} C_VEL
LIN {X 0,Y 660.419,Z 918.745,A -85,B 0,C 180,E1 30188.925,E2 30188.925} C_VEL
LIN {X 0,Y 658.812,Z 940.779,A -85,B 0,C 180,E1 30188.029,E2 30188.029} C_VEL
LIN {X 0,Y 657.097,Z 962.82,A -85,B 0,C 180,E1 30186.994,E2 30186.994} C_VEL
LIN {X 0,Y 654.914,Z 988.961,A -85,B 0,C 180,E1 30185.568,E2 30185.568} C_VEL
LIN {X 0,Y 652.994,Z 1010.384,A -85,B 0,C 180,E1 30184.221,E2 30184.221} C_VEL
LIN {X 0,Y 651.254,Z 1029.469,A -85,B 0,C 180,E1 30182.878,E2 30182.878} C_VEL
LIN {X 0,Y 649.322,Z 1051.289,A -85,B 0,C 180,E1 30181.157,E2 30181.157} C_VEL
LIN {X 0,Y 647.517,Z 1071.281,A -85,B 0,C 180,E1 30179.358,E2 30179.358} C_VEL
LIN {X 0,Y 646.096,Z 1087.698,A -85,B 0,C 180,E1 30177.721,E2 30177.721} C_VEL
LIN {X 0,Y 644.596,Z 1106.401,A -85,B 0,C 180,E1 30175.643,E2 30175.643} C_VEL
LIN {X 0,Y 643.323,Z 1122.988,A -85,B 0,C 180,E1 30173.543,E2 30173.543} C_VEL
LIN {X 0,Y 642.423,Z 1136.384,A -85,B 0,C 180,E1 30171.646,E2 30171.646} C_VEL
LIN {X 0,Y 641.561,Z 1151.099,A -85,B 0,C 180,E1 30169.293,E2 30169.293} C_VEL
LIN {X 0,Y 640.932,Z 1163.146,A -85,B 0,C 180,E1 30167.055,E2 30167.055} C_VEL
LIN {X 0,Y 640.55,Z 1172.309,A -85,B 0,C 180,E1 30165.11,E2 30165.11} C_VEL
LIN {X 0,Y 640.289,Z 1180.578,A -85,B 0,C 180,E1 30163.087,E2 30163.087} C_VEL
LIN {X 0,Y 640.073,Z 1188.478,A -85,B 0,C 180,E1 30160.804,E2 30160.804} C_VEL
LIN {X 0,Y 639.978,Z 1195.12,A -85,B 0,C 180,E1 30158.355,E2 30158.355} C_VEL
LIN {X 0,Y 639.931,Z 1199.724,A -85,B 0,C 180,E1 30156.099,E2 30156.099} C_VEL
LIN {X 0,Y 639.912,Z 1203.094,A -85,B 0,C 180,E1 30153.673,E2 30153.673} C_VEL
LIN {X 0,Y 639.914,Z 1204.669,A -85,B 0,C 180,E1 30151.343,E2 30151.343} C_VEL
LIN {X 0,Y 639.894,Z 1204.849,A -85,B 0,C 180,E1 30149.373,E2 30149.373} C_VEL
LIN {X 0,Y 639.91,Z 1203.941,A -85,B 0,C 180,E1 30147.313,E2 30147.313} C_VEL
LIN {X 0,Y 639.922,Z 1201.552,A -85,B 0,C 180,E1 30145.07,E2 30145.07} C_VEL
LIN {X 0,Y 639.953,Z 1197.347,A -85,B 0,C 180,E1 30142.639,E2 30142.639} C_VEL
LIN {X 0,Y 640.026,Z 1191.624,A -85,B 0,C 180,E1 30140.287,E2 30140.287} C_VEL
LIN {X 0,Y 640.164,Z 1184.591,A -85,B 0,C 180,E1 30138.011,E2 30138.011} C_VEL
LIN {X 0,Y 640.484,Z 1174.741,A -85,B 0,C 180,E1 30135.443,E2 30135.443} C_VEL
LIN {X 0,Y 640.843,Z 1165.002,A -85,B 0,C 180,E1 30133.317,E2 30133.317} C_VEL
LIN {X 0,Y 641.352,Z 1154.761,A -85,B 0,C 180,E1 30131.362,E2 30131.362} C_VEL
LIN {X 0,Y 642.053,Z 1142.531,A -85,B 0,C 180,E1 30129.298,E2 30129.298} C_VEL
LIN {X 0,Y 643.082,Z 1126.501,A -85,B 0,C 180,E1 30126.933,E2 30126.933} C_VEL
LIN {X 0,Y 644.144,Z 1111.859,A -85,B 0,C 180,E1 30125.026,E2 30125.026} C_VEL
LIN {X 0,Y 645.467,Z 1095.435,A -85,B 0,C 180,E1 30123.107,E2 30123.107} C_VEL
LIN {X 0,Y 647.156,Z 1075.337,A -85,B 0,C 180,E1 30121.03,E2 30121.03} C_VEL
LIN {X 0,Y 648.61,Z 1058.942,A -85,B 0,C 180,E1 30119.514,E2 30119.514} C_VEL
LIN {X 0,Y 650.17,Z 1041.626,A -85,B 0,C 180,E1 30118.061,E2 30118.061} C_VEL
LIN {X 0,Y 652.2,Z 1019.55,A -85,B 0,C 180,E1 30116.397,E2 30116.397} C_VEL
LIN {X 0,Y 654.232,Z 996.179,A -85,B 0,C 180,E1 30114.867,E2 30114.867} C_VEL
LIN {X 0,Y 655.998,Z 975.858,A -85,B 0,C 180,E1 30113.691,E2 30113.691} C_VEL
LIN {X 0,Y 657.988,Z 952.264,A -85,B 0,C 180,E1 30112.49,E2 30112.49} C_VEL
LIN {X 0,Y 659.917,Z 926.451,A -85,B 0,C 180,E1 30111.374,E2 30111.374} C_VEL
LIN {X 0,Y 661.329,Z 904.877,A -85,B 0,C 180,E1 30110.581,E2 30110.581} C_VEL
LIN {X 0,Y 662.652,Z 883.013,A -85,B 0,C 180,E1 30109.901,E2 30109.901} C_VEL
LIN {X 0,Y 663.946,Z 858.265,A -85,B 0,C 180,E1 30109.275,E2 30109.275} C_VEL
LIN {X 0,Y 665.052,Z 829.746,A -85,B 0,C 180,E1 30108.74,E2 30108.74} C_VEL
LIN {X 0,Y 666.541,Z 746.819,A -85,B 0,C 180,E1 30107.644,E2 30107.644} C_VEL
LIN {X 0,Y 670.245,Z 524.663,A -85,B 0,C 180,E1 30104.707,E2 30104.707} C_VEL
LIN {X 0,Y 672.691,Z 379.682,A -85,B 0,C 180,E1 30102.728,E2 30102.728} C_VEL
LIN {X 0,Y 666.118,Z 349.426,A -85,B 0,C 180,E1 30101.681,E2 30101.681} C_VEL
LIN {X 0,Y 655.476,Z 328.548,A -85,B 0,C 180,E1 30099.204,E2 30099.204} C_VEL
LIN {X 0,Y 649.028,Z 315.909,A -85,B 0,C 180,E1 30097.595,E2 30097.595} C_VEL
LIN {X 0,Y 644.505,Z 307.307,A -85,B 0,C 180,E1 30096.455,E2 30096.455} C_VEL
LIN {X 0,Y 642.868,Z 303.88,A -85,B 0,C 180,E1 30096.01,E2 30096.01} C_VEL
LIN {X 0,Y 641.123,Z 300.81,A -85,B 0,C 180,E1 30095.572,E2 30095.572} C_VEL
LIN {X 0,Y 640.85,Z 299.574,A -85,B 0,C 180,E1 30095.37,E2 30095.37} C_VEL
LIN {X 0,Y 640.813,Z 299.377,A -85,B 0,C 180,E1 30092.146,E2 30092.146} C_VEL
LIN {X 0,Y 640.822,Z 299.409,A -85,B 0,C 180,E1 30089.03,E2 30089.03} C_VEL
LIN {X 0,Y 640.812,Z 299.382,A -85,B 0,C 180,E1 30085.906,E2 30085.906} C_VEL
LIN {X 0,Y 640.816,Z 299.385,A -85,B 0,C 180,E1 30082.863,E2 30082.863} C_VEL
LIN {X 0,Y 640.818,Z 299.398,A -85,B 0,C 180,E1 30079.791,E2 30079.791} C_VEL
LIN {X 0,Y 640.81,Z 299.371,A -85,B 0,C 180,E1 30076.66,E2 30076.66} C_VEL
LIN {X 0,Y 640.816,Z 299.4,A -85,B 0,C 180,E1 30073.536,E2 30073.536} C_VEL
LIN {X 0,Y 640.808,Z 299.372,A -85,B 0,C 180,E1 30070.519,E2 30070.519} C_VEL
LIN {X 0,Y 640.82,Z 299.394,A -85,B 0,C 180,E1 30067.441,E2 30067.441} C_VEL
LIN {X 0,Y 640.809,Z 299.401,A -85,B 0,C 180,E1 30064.385,E2 30064.385} C_VEL
LIN {X 0,Y 640.825,Z 299.399,A -85,B 0,C 180,E1 30061.341,E2 30061.341} C_VEL
LIN {X 0,Y 640.805,Z 299.399,A -85,B 0,C 180,E1 30058.212,E2 30058.212} C_VEL
LIN {X 0,Y 640.825,Z 299.404,A -85,B 0,C 180,E1 30055.167,E2 30055.167} C_VEL
LIN {X 0,Y 640.803,Z 299.409,A -85,B 0,C 180,E1 30052.108,E2 30052.108} C_VEL
LIN {X 0,Y 640.827,Z 299.401,A -85,B 0,C 180,E1 30049.026,E2 30049.026} C_VEL
LIN {X 0,Y 640.798,Z 299.409,A -85,B 0,C 180,E1 30045.911,E2 30045.911} C_VEL
LIN {X 0,Y 640.828,Z 299.394,A -85,B 0,C 180,E1 30042.848,E2 30042.848} C_VEL
LIN {X 0,Y 640.794,Z 299.401,A -85,B 0,C 180,E1 30039.732,E2 30039.732} C_VEL
LIN {X 0,Y 640.831,Z 299.399,A -85,B 0,C 180,E1 30036.749,E2 30036.749} C_VEL
LIN {X 0,Y 640.791,Z 299.384,A -85,B 0,C 180,E1 30033.591,E2 30033.591} C_VEL
LIN {X 0,Y 640.832,Z 299.401,A -85,B 0,C 180,E1 30030.561,E2 30030.561} C_VEL
LIN {X 0,Y 640.789,Z 299.384,A -85,B 0,C 180,E1 30027.535,E2 30027.535} C_VEL
LIN {X 0,Y 640.825,Z 299.395,A -85,B 0,C 180,E1 30024.518,E2 30024.518} C_VEL
LIN {X 0,Y 640.785,Z 299.399,A -85,B 0,C 180,E1 30021.379,E2 30021.379} C_VEL
LIN {X 0,Y 640.812,Z 299.377,A -85,B 0,C 180,E1 30018.459,E2 30018.459} C_VEL
LIN {X 0,Y 640.786,Z 299.408,A -85,B 0,C 180,E1 30015.271,E2 30015.271} C_VEL
LIN {X 0,Y 640.811,Z 299.381,A -85,B 0,C 180,E1 30014.367,E2 30014.367} C_VEL
LIN {X 0,Y 639.829,Z 299.496,A -85,B 0,C 180,E1 30013.908,E2 30013.908} C_VEL
LIN {X 0,Y 633.609,Z 300.272,A -85,B 0,C 180,E1 30012.733,E2 30012.733} C_VEL
LIN {X 0,Y 632.869,Z 300.373,A -85,B 0,C 180,E1 30012.331,E2 30012.331} C_VEL
LIN {X 0,Y 632.918,Z 300.76,A -85,B 0,C 180,E1 30011.408,E2 30011.408} C_VEL
LIN {X 0,Y 634.193,Z 303.956,A -85,B 0,C 180,E1 30010.956,E2 30010.956} C_VEL
LIN {X 0,Y 637.706,Z 311.032,A -85,B 0,C 180,E1 30009.939,E2 30009.939} C_VEL
LIN {X 0,Y 645.037,Z 326.069,A -85,B 0,C 180,E1 30007.867,E2 30007.867} C_VEL
LIN {X 0,Y 652.228,Z 342.086,A -85,B 0,C 180,E1 30005.808,E2 30005.808} C_VEL
LIN {X 0,Y 654.618,Z 347.557,A -85,B 0,C 180,E1 30005.174,E2 30005.174} C_VEL
LIN {X 0,Y 656.65,Z 355.127,A -85,B 0,C 180,E1 30004.869,E2 30004.869} C_VEL
LIN {X 0,Y 661.767,Z 378.516,A -85,B 0,C 180,E1 30004.054,E2 30004.054} C_VEL
LIN {X 0,Y 657.216,Z 618.538,A -85,B 0,C 180,E1 30000.886,E2 30000.886} C_VEL
LIN {X 0,Y 654.27,Z 782.474,A -85,B 0,C 180,E1 29998.748,E2 29998.748} C_VEL
LIN {X 0,Y 653.286,Z 808.983,A -85,B 0,C 180,E1 29998.249,E2 29998.249} C_VEL
LIN {X 0,Y 652.241,Z 830.047,A -85,B 0,C 180,E1 29997.723,E2 29997.723} C_VEL
LIN {X 0,Y 651.129,Z 849.472,A -85,B 0,C 180,E1 29997.133,E2 29997.133} C_VEL
LIN {X 0,Y 649.749,Z 871.01,A -85,B 0,C 180,E1 29996.356,E2 29996.356} C_VEL
LIN {X 0,Y 647.884,Z 896.344,A -85,B 0,C 180,E1 29995.259,E2 29995.259} C_VEL
LIN {X 0,Y 646.219,Z 917.03,A -85,B 0,C 180,E1 29994.206,E2 29994.206} C_VEL
LIN {X 0,Y 644.349,Z 939.842,A -85,B 0,C 180,E1 29992.874,E2 29992.874} C_VEL
LIN {X 0,Y 642.441,Z 961.406,A -85,B 0,C 180,E1 29991.405,E2 29991.405} C_VEL
LIN {X 0,Y 640.843,Z 979.401,A -85,B 0,C 180,E1 29990.027,E2 29990.027} C_VEL
LIN {X 0,Y 639.044,Z 1000.067,A -85,B 0,C 180,E1 29988.235,E2 29988.235} C_VEL
LIN {X 0,Y 637.623,Z 1016.838,A -85,B 0,C 180,E1 29986.582,E2 29986.582} C_VEL
LIN {X 0,Y 636.268,Z 1033.52,A -85,B 0,C 180,E1 29984.748,E2 29984.748} C_VEL
LIN {X 0,Y 635.076,Z 1049.545,A -85,B 0,C 180,E1 29982.733,E2 29982.733} C_VEL
LIN {X 0,Y 634.188,Z 1062.433,A -85,B 0,C 180,E1 29980.906,E2 29980.906} C_VEL
LIN {X 0,Y 633.393,Z 1076.046,A -85,B 0,C 180,E1 29978.716,E2 29978.716} C_VEL
LIN {X 0,Y 632.828,Z 1087.187,A -85,B 0,C 180,E1 29976.623,E2 29976.623} C_VEL
LIN {X 0,Y 632.478,Z 1096.011,A -85,B 0,C 180,E1 29974.715,E2 29974.715} C_VEL
LIN {X 0,Y 632.19,Z 1105.251,A -85,B 0,C 180,E1 29972.357,E2 29972.357} C_VEL
LIN {X 0,Y 632.033,Z 1112.052,A -85,B 0,C 180,E1 29970.181,E2 29970.181} C_VEL
LIN {X 0,Y 631.954,Z 1116.834,A -85,B 0,C 180,E1 29968.277,E2 29968.277} C_VEL
LIN {X 0,Y 631.923,Z 1120.998,A -85,B 0,C 180,E1 29966.099,E2 29966.099} C_VEL
LIN {X 0,Y 631.917,Z 1123.761,A -85,B 0,C 180,E1 29963.732,E2 29963.732} C_VEL
LIN {X 0,Y 631.915,Z 1124.795,A -85,B 0,C 180,E1 29961.813,E2 29961.813} C_VEL
LIN {X 0,Y 631.901,Z 1124.742,A -85,B 0,C 180,E1 29959.884,E2 29959.884} C_VEL
LIN {X 0,Y 631.916,Z 1123.184,A -85,B 0,C 180,E1 29957.499,E2 29957.499} C_VEL
LIN {X 0,Y 631.917,Z 1120.163,A -85,B 0,C 180,E1 29955.335,E2 29955.335} C_VEL
LIN {X 0,Y 631.967,Z 1116.429,A -85,B 0,C 180,E1 29953.454,E2 29953.454} C_VEL
LIN {X 0,Y 632.05,Z 1111.304,A -85,B 0,C 180,E1 29951.46,E2 29951.46} C_VEL
LIN {X 0,Y 632.236,Z 1103.453,A -85,B 0,C 180,E1 29949.059,E2 29949.059} C_VEL
LIN {X 0,Y 632.503,Z 1095.234,A -85,B 0,C 180,E1 29947.017,E2 29947.017} C_VEL
LIN {X 0,Y 632.898,Z 1086.014,A -85,B 0,C 180,E1 29945.051,E2 29945.051} C_VEL
LIN {X 0,Y 633.568,Z 1072.887,A -85,B 0,C 180,E1 29942.662,E2 29942.662} C_VEL
LIN {X 0,Y 634.308,Z 1060.71,A -85,B 0,C 180,E1 29940.748,E2 29940.748} C_VEL
LIN {X 0,Y 635.333,Z 1046.089,A -85,B 0,C 180,E1 29938.712,E2 29938.712} C_VEL
LIN {X 0,Y 636.555,Z 1029.95,A -85,B 0,C 180,E1 29936.757,E2 29936.757} C_VEL
LIN {X 0,Y 637.794,Z 1014.607,A -85,B 0,C 180,E1 29935.096,E2 29935.096} C_VEL
LIN {X 0,Y 639.485,Z 995.031,A -85,B 0,C 180,E1 29933.214,E2 29933.214} C_VEL
LIN {X 0,Y 641.083,Z 976.819,A -85,B 0,C 180,E1 29931.677,E2 29931.677} C_VEL
LIN {X 0,Y 642.68,Z 958.718,A -85,B 0,C 180,E1 29930.309,E2 29930.309} C_VEL
LIN {X 0,Y 644.684,Z 935.412,A -85,B 0,C 180,E1 29928.765,E2 29928.765} C_VEL
LIN {X 0,Y 646.306,Z 916.029,A -85,B 0,C 180,E1 29927.65,E2 29927.65} C_VEL
LIN {X 0,Y 648.009,Z 894.893,A -85,B 0,C 180,E1 29926.582,E2 29926.582} C_VEL
LIN {X 0,Y 649.827,Z 869.738,A -85,B 0,C 180,E1 29925.504,E2 29925.504} C_VEL
LIN {X 0,Y 651.174,Z 848.744,A -85,B 0,C 180,E1 29924.753,E2 29924.753} C_VEL
LIN {X 0,Y 652.349,Z 828.052,A -85,B 0,C 180,E1 29924.131,E2 29924.131} C_VEL
LIN {X 0,Y 653.544,Z 802.45,A -85,B 0,C 180,E1 29923.517,E2 29923.517} C_VEL
LIN {X 0,Y 654.359,Z 778.093,A -85,B 0,C 180,E1 29923.098,E2 29923.098} C_VEL
LIN {X 0,Y 658.834,Z 536.073,A -85,B 0,C 180,E1 29919.935,E2 29919.935} C_VEL
LIN {X 0,Y 661.793,Z 377.209,A -85,B 0,C 180,E1 29917.81,E2 29917.81} C_VEL
LIN {X 0,Y 655.451,Z 349.389,A -85,B 0,C 180,E1 29916.802,E2 29916.802} C_VEL
LIN {X 0,Y 654.409,Z 346.944,A -85,B 0,C 180,E1 29916.652,E2 29916.652} C_VEL
LIN {X 0,Y 648.202,Z 332.499,A -85,B 0,C 180,E1 29914.803,E2 29914.803} C_VEL
LIN {X 0,Y 641.5,Z 318.032,A -85,B 0,C 180,E1 29912.742,E2 29912.742} C_VEL
LIN {X 0,Y 636.896,Z 308.91,A -85,B 0,C 180,E1 29911.309,E2 29911.309} C_VEL
LIN {X 0,Y 634.681,Z 304.549,A -85,B 0,C 180,E1 29910.588,E2 29910.588} C_VEL
LIN {X 0,Y 632.937,Z 300.76,A -85,B 0,C 180,E1 29909.951,E2 29909.951} C_VEL
LIN {X 0,Y 632.877,Z 300.366,A -85,B 0,C 180,E1 29909.113,E2 29909.113} C_VEL
LIN {X 0,Y 632.882,Z 300.363,A -85,B 0,C 180,E1 29905.953,E2 29905.953} C_VEL
LIN {X 0,Y 632.875,Z 300.382,A -85,B 0,C 180,E1 29902.871,E2 29902.871} C_VEL
LIN {X 0,Y 632.883,Z 300.394,A -85,B 0,C 180,E1 29899.761,E2 29899.761} C_VEL
LIN {X 0,Y 632.869,Z 300.361,A -85,B 0,C 180,E1 29896.617,E2 29896.617} C_VEL
LIN {X 0,Y 632.878,Z 300.382,A -85,B 0,C 180,E1 29893.523,E2 29893.523} C_VEL
LIN {X 0,Y 632.872,Z 300.388,A -85,B 0,C 180,E1 29890.376,E2 29890.376} C_VEL
LIN {X 0,Y 632.872,Z 300.361,A -85,B 0,C 180,E1 29887.353,E2 29887.353} C_VEL
LIN {X 0,Y 632.876,Z 300.395,A -85,B 0,C 180,E1 29884.259,E2 29884.259} C_VEL
LIN {X 0,Y 632.872,Z 300.363,A -85,B 0,C 180,E1 29881.177,E2 29881.177} C_VEL
LIN {X 0,Y 632.877,Z 300.395,A -85,B 0,C 180,E1 29878.099,E2 29878.099} C_VEL
LIN {X 0,Y 632.872,Z 300.371,A -85,B 0,C 180,E1 29875.015,E2 29875.015} C_VEL
LIN {X 0,Y 632.875,Z 300.379,A -85,B 0,C 180,E1 29871.917,E2 29871.917} C_VEL
LIN {X 0,Y 632.87,Z 300.391,A -85,B 0,C 180,E1 29868.794,E2 29868.794} C_VEL
LIN {X 0,Y 632.875,Z 300.364,A -85,B 0,C 180,E1 29865.731,E2 29865.731} C_VEL
LIN {X 0,Y 632.87,Z 300.396,A -85,B 0,C 180,E1 29862.626,E2 29862.626} C_VEL
LIN {X 0,Y 632.876,Z 300.367,A -85,B 0,C 180,E1 29859.531,E2 29859.531} C_VEL
LIN {X 0,Y 632.866,Z 300.374,A -85,B 0,C 180,E1 29856.538,E2 29856.538} C_VEL
LIN {X 0,Y 632.882,Z 300.397,A -85,B 0,C 180,E1 29853.405,E2 29853.405} C_VEL
LIN {X 0,Y 632.865,Z 300.374,A -85,B 0,C 180,E1 29850.336,E2 29850.336} C_VEL
LIN {X 0,Y 632.885,Z 300.399,A -85,B 0,C 180,E1 29847.294,E2 29847.294} C_VEL
LIN {X 0,Y 632.926,Z 300.687,A -85,B 0,C 180,E1 29845.619,E2 29845.619} C_VEL
LIN {X 0,Y 634.299,Z 304.04,A -85,B 0,C 180,E1 29845.094,E2 29845.094} C_VEL
LIN {X 0,Y 635.653,Z 306.156,A -85,B 0,C 180,E1 29844.739,E2 29844.739} C_VEL
LIN {X 0,Y 640.77,Z 315.931,A -85,B 0,C 180,E1 29843.298,E2 29843.298} C_VEL
LIN {X 0,Y 647.409,Z 329.056,A -85,B 0,C 180,E1 29841.537,E2 29841.537} C_VEL
LIN {X 0,Y 658.208,Z 350.291,A -85,B 0,C 180,E1 29838.985,E2 29838.985} C_VEL
LIN {X 0,Y 661.013,Z 354.747,A -85,B 0,C 180,E1 29838.657,E2 29838.657} C_VEL
LIN {X 0,Y 667.087,Z 383.017,A -85,B 0,C 180,E1 29837.699,E2 29837.699} C_VEL
LIN {X 0,Y 663.987,Z 558.549,A -85,B 0,C 180,E1 29835.328,E2 29835.328} C_VEL
LIN {X 0,Y 659.969,Z 785.031,A -85,B 0,C 180,E1 29832.325,E2 29832.325} C_VEL
LIN {X 0,Y 658.933,Z 833.382,A -85,B 0,C 180,E1 29831.665,E2 29831.665} C_VEL
LIN {X 0,Y 657.695,Z 860.938,A -85,B 0,C 180,E1 29831.121,E2 29831.121} C_VEL
LIN {X 0,Y 656.409,Z 884.032,A -85,B 0,C 180,E1 29830.525,E2 29830.525} C_VEL
LIN {X 0,Y 654.997,Z 905.877,A -85,B 0,C 180,E1 29829.838,E2 29829.838} C_VEL
LIN {X 0,Y 653.195,Z 931.532,A -85,B 0,C 180,E1 29828.873,E2 29828.873} C_VEL
LIN {X 0,Y 651.038,Z 956.888,A -85,B 0,C 180,E1 29827.724,E2 29827.724} C_VEL
LIN {X 0,Y 649.169,Z 977.835,A -85,B 0,C 180,E1 29826.632,E2 29826.632} C_VEL
LIN {X 0,Y 647.122,Z 999.846,A -85,B 0,C 180,E1 29825.33,E2 29825.33} C_VEL
LIN {X 0,Y 644.786,Z 1024.238,A -85,B 0,C 180,E1 29823.667,E2 29823.667} C_VEL
LIN {X 0,Y 642.956,Z 1042.842,A -85,B 0,C 180,E1 29822.235,E2 29822.235} C_VEL
LIN {X 0,Y 641.224,Z 1060.72,A -85,B 0,C 180,E1 29820.708,E2 29820.708} C_VEL
LIN {X 0,Y 639.241,Z 1081.498,A -85,B 0,C 180,E1 29818.724,E2 29818.724} C_VEL
LIN {X 0,Y 637.683,Z 1098.847,A -85,B 0,C 180,E1 29816.845,E2 29816.845} C_VEL
LIN {X 0,Y 636.315,Z 1114.602,A -85,B 0,C 180,E1 29814.948,E2 29814.948} C_VEL
LIN {X 0,Y 634.989,Z 1131.894,A -85,B 0,C 180,E1 29812.594,E2 29812.594} C_VEL
LIN {X 0,Y 634.107,Z 1144.859,A -85,B 0,C 180,E1 29810.587,E2 29810.587} C_VEL
LIN {X 0,Y 633.407,Z 1156.309,A -85,B 0,C 180,E1 29808.594,E2 29808.594} C_VEL
LIN {X 0,Y 632.814,Z 1168.202,A -85,B 0,C 180,E1 29806.24,E2 29806.24} C_VEL
LIN {X 0,Y 632.401,Z 1178.185,A -85,B 0,C 180,E1 29803.88,E2 29803.88} C_VEL
LIN {X 0,Y 632.166,Z 1185.9,A -85,B 0,C 180,E1 29801.743,E2 29801.743} C_VEL
LIN {X 0,Y 632.021,Z 1192.865,A -85,B 0,C 180,E1 29799.378,E2 29799.378} C_VEL
LIN {X 0,Y 631.94,Z 1198.422,A -85,B 0,C 180,E1 29796.906,E2 29796.906} C_VEL
LIN {X 0,Y 631.913,Z 1202.016,A -85,B 0,C 180,E1 29794.629,E2 29794.629} C_VEL
LIN {X 0,Y 631.91,Z 1204.211,A -85,B 0,C 180,E1 29792.358,E2 29792.358} C_VEL
LIN {X 0,Y 631.902,Z 1204.961,A -85,B 0,C 180,E1 29789.819,E2 29789.819} C_VEL
LIN {X 0,Y 631.908,Z 1204.075,A -85,B 0,C 180,E1 29787.461,E2 29787.461} C_VEL
LIN {X 0,Y 631.917,Z 1201.788,A -85,B 0,C 180,E1 29785.19,E2 29785.19} C_VEL
LIN {X 0,Y 631.957,Z 1197.735,A -85,B 0,C 180,E1 29782.728,E2 29782.728} C_VEL
LIN {X 0,Y 632.034,Z 1191.876,A -85,B 0,C 180,E1 29780.255,E2 29780.255} C_VEL
LIN {X 0,Y 632.182,Z 1184.891,A -85,B 0,C 180,E1 29777.95,E2 29777.95} C_VEL
LIN {X 0,Y 632.529,Z 1175.145,A -85,B 0,C 180,E1 29775.35,E2 29775.35} C_VEL
LIN {X 0,Y 632.943,Z 1165,A -85,B 0,C 180,E1 29773.102,E2 29773.102} C_VEL
LIN {X 0,Y 633.497,Z 1154.763,A -85,B 0,C 180,E1 29771.122,E2 29771.122} C_VEL
LIN {X 0,Y 634.299,Z 1141.951,A -85,B 0,C 180,E1 29768.937,E2 29768.937} C_VEL
LIN {X 0,Y 635.434,Z 1125.799,A -85,B 0,C 180,E1 29766.541,E2 29766.541} C_VEL
LIN {X 0,Y 636.63,Z 1111.083,A -85,B 0,C 180,E1 29764.611,E2 29764.611} C_VEL
LIN {X 0,Y 638.206,Z 1092.836,A -85,B 0,C 180,E1 29762.47,E2 29762.47} C_VEL
LIN {X 0,Y 639.969,Z 1073.816,A -85,B 0,C 180,E1 29760.519,E2 29760.519} C_VEL
LIN {X 0,Y 641.533,Z 1057.513,A -85,B 0,C 180,E1 29759.007,E2 29759.007} C_VEL
LIN {X 0,Y 643.319,Z 1039.19,A -85,B 0,C 180,E1 29757.469,E2 29757.469} C_VEL
LIN {X 0,Y 645.642,Z 1015.192,A -85,B 0,C 180,E1 29755.688,E2 29755.688} C_VEL
LIN {X 0,Y 647.617,Z 994.635,A -85,B 0,C 180,E1 29754.351,E2 29754.351} C_VEL
LIN {X 0,Y 649.503,Z 974.414,A -85,B 0,C 180,E1 29753.181,E2 29753.181} C_VEL
LIN {X 0,Y 651.752,Z 949.299,A -85,B 0,C 180,E1 29751.909,E2 29751.909} C_VEL
LIN {X 0,Y 653.674,Z 924.585,A -85,B 0,C 180,E1 29750.854,E2 29750.854} C_VEL
LIN {X 0,Y 655.115,Z 904.134,A -85,B 0,C 180,E1 29750.104,E2 29750.104} C_VEL
LIN {X 0,Y 656.512,Z 882.384,A -85,B 0,C 180,E1 29749.428,E2 29749.428} C_VEL
LIN {X 0,Y 657.914,Z 857.27,A -85,B 0,C 180,E1 29748.794,E2 29748.794} C_VEL
LIN {X 0,Y 659.041,Z 829.29,A -85,B 0,C 180,E1 29748.273,E2 29748.273} C_VEL
LIN {X 0,Y 660.725,Z 740.972,A -85,B 0,C 180,E1 29747.097,E2 29747.097} C_VEL
LIN {X 0,Y 664.716,Z 519.358,A -85,B 0,C 180,E1 29744.143,E2 29744.143} C_VEL
LIN {X 0,Y 666.994,Z 381.732,A -85,B 0,C 180,E1 29742.27,E2 29742.27} C_VEL
LIN {X 0,Y 660.71,Z 353.832,A -85,B 0,C 180,E1 29741.287,E2 29741.287} C_VEL
LIN {X 0,Y 657.792,Z 349.472,A -85,B 0,C 180,E1 29740.931,E2 29740.931} C_VEL
LIN {X 0,Y 645.65,Z 325.51,A -85,B 0,C 180,E1 29737.979,E2 29737.979} C_VEL
LIN {X 0,Y 638.892,Z 312.644,A -85,B 0,C 180,E1 29736.27,E2 29736.27} C_VEL
LIN {X 0,Y 636.8,Z 308.724,A -85,B 0,C 180,E1 29735.732,E2 29735.732} C_VEL
LIN {X 0,Y 634.448,Z 304.237,A -85,B 0,C 180,E1 29735.117,E2 29735.117} C_VEL
LIN {X 0,Y 632.92,Z 300.624,A -85,B 0,C 180,E1 29734.604,E2 29734.604} C_VEL
LIN {X 0,Y 632.873,Z 300.357,A -85,B 0,C 180,E1 29731.531,E2 29731.531} C_VEL
LIN {X 0,Y 632.893,Z 300.384,A -85,B 0,C 180,E1 29728.363,E2 29728.363} C_VEL
LIN {X 0,Y 632.886,Z 300.384,A -85,B 0,C 180,E1 29725.144,E2 29725.144} C_VEL
LIN {X 0,Y 632.879,Z 300.356,A -85,B 0,C 180,E1 29721.892,E2 29721.892} C_VEL
LIN {X 0,Y 632.881,Z 300.398,A -85,B 0,C 180,E1 29718.802,E2 29718.802} C_VEL
LIN {X 0,Y 632.875,Z 300.35,A -85,B 0,C 180,E1 29715.674,E2 29715.674} C_VEL
LIN {X 0,Y 632.875,Z 300.395,A -85,B 0,C 180,E1 29712.593,E2 29712.593} C_VEL
LIN {X 0,Y 632.874,Z 300.349,A -85,B 0,C 180,E1 29709.457,E2 29709.457} C_VEL
LIN {X 0,Y 632.87,Z 300.396,A -85,B 0,C 180,E1 29706.35,E2 29706.35} C_VEL
LIN {X 0,Y 632.882,Z 300.391,A -85,B 0,C 180,E1 29703.261,E2 29703.261} C_VEL
LIN {X 0,Y 632.866,Z 300.397,A -85,B 0,C 180,E1 29700.181,E2 29700.181} C_VEL
LIN {X 0,Y 632.882,Z 300.383,A -85,B 0,C 180,E1 29697.102,E2 29697.102} C_VEL
LIN {X 0,Y 632.861,Z 300.387,A -85,B 0,C 180,E1 29694.014,E2 29694.014} C_VEL
LIN {X 0,Y 632.889,Z 300.393,A -85,B 0,C 180,E1 29691.001,E2 29691.001} C_VEL
LIN {X 0,Y 632.859,Z 300.393,A -85,B 0,C 180,E1 29687.87,E2 29687.87} C_VEL
LIN {X 0,Y 632.888,Z 300.394,A -85,B 0,C 180,E1 29684.796,E2 29684.796} C_VEL
LIN {X 0,Y 632.855,Z 300.398,A -85,B 0,C 180,E1 29681.674,E2 29681.674} C_VEL
LIN {X 0,Y 632.89,Z 300.39,A -85,B 0,C 180,E1 29678.595,E2 29678.595} C_VEL
LIN {X 0,Y 632.848,Z 300.362,A -85,B 0,C 180,E1 29675.546,E2 29675.546} C_VEL
LIN {X 0,Y 632.892,Z 300.386,A -85,B 0,C 180,E1 29672.425,E2 29672.425} C_VEL
LIN {X 0,Y 632.845,Z 300.367,A -85,B 0,C 180,E1 29669.419,E2 29669.419} C_VEL
LIN {X 0,Y 632.892,Z 300.389,A -85,B 0,C 180,E1 29666.321,E2 29666.321} C_VEL
LIN {X 0,Y 632.84,Z 300.359,A -85,B 0,C 180,E1 29663.229,E2 29663.229} C_VEL
LIN {X 0,Y 632.895,Z 300.398,A -85,B 0,C 180,E1 29660.156,E2 29660.156} C_VEL
LIN {X 0,Y 632.838,Z 300.372,A -85,B 0,C 180,E1 29657.079,E2 29657.079} C_VEL
LIN {X 0,Y 632.89,Z 300.359,A -85,B 0,C 180,E1 29654.04,E2 29654.04} C_VEL
LIN {X 0,Y 632.869,Z 300.373,A -85,B 0,C 180,E1 29652.331,E2 29652.331} C_VEL
LIN {X 0,Y 632.457,Z 301.31,A -85,B 0,C 180,E1 29651.94,E2 29651.94} C_VEL
LIN {X 0,Y 631.181,Z 304.426,A -85,B 0,C 180,E1 29651.482,E2 29651.482} C_VEL
LIN {X 0,Y 629.851,Z 310.103,A -85,B 0,C 180,E1 29650.903,E2 29650.903} C_VEL
LIN {X 0,Y 630.45,Z 313.328,A -85,B 0,C 180,E1 29650.512,E2 29650.512} C_VEL
LIN {X 0,Y 638.968,Z 330.846,A -85,B 0,C 180,E1 29648.063,E2 29648.063} C_VEL
LIN {X 0,Y 646.236,Z 347.014,A -85,B 0,C 180,E1 29645.98,E2 29645.98} C_VEL
LIN {X 0,Y 650.16,Z 353.377,A -85,B 0,C 180,E1 29645.498,E2 29645.498} C_VEL
LIN {X 0,Y 656.122,Z 380.057,A -85,B 0,C 180,E1 29644.533,E2 29644.533} C_VEL
LIN {X 0,Y 651.291,Z 619.673,A -85,B 0,C 180,E1 29641.348,E2 29641.348} C_VEL
LIN {X 0,Y 648.133,Z 780.816,A -85,B 0,C 180,E1 29639.226,E2 29639.226} C_VEL
LIN {X 0,Y 647.056,Z 807.689,A -85,B 0,C 180,E1 29638.723,E2 29638.723} C_VEL
LIN {X 0,Y 645.761,Z 831.418,A -85,B 0,C 180,E1 29638.12,E2 29638.12} C_VEL
LIN {X 0,Y 644.188,Z 856.453,A -85,B 0,C 180,E1 29637.325,E2 29637.325} C_VEL
LIN {X 0,Y 642.378,Z 880.559,A -85,B 0,C 180,E1 29636.384,E2 29636.384} C_VEL
LIN {X 0,Y 640.758,Z 900.665,A -85,B 0,C 180,E1 29635.461,E2 29635.461} C_VEL
LIN {X 0,Y 638.841,Z 923.429,A -85,B 0,C 180,E1 29634.258,E2 29634.258} C_VEL
LIN {X 0,Y 636.785,Z 945.739,A -85,B 0,C 180,E1 29632.874,E2 29632.874} C_VEL
LIN {X 0,Y 635.099,Z 963.678,A -85,B 0,C 180,E1 29631.617,E2 29631.617} C_VEL
LIN {X 0,Y 633.17,Z 984.077,A -85,B 0,C 180,E1 29630.012,E2 29630.012} C_VEL
LIN {X 0,Y 631.355,Z 1003.253,A -85,B 0,C 180,E1 29628.274,E2 29628.274} C_VEL
LIN {X 0,Y 629.867,Z 1019.755,A -85,B 0,C 180,E1 29626.603,E2 29626.603} C_VEL
LIN {X 0,Y 628.262,Z 1038.294,A -85,B 0,C 180,E1 29624.469,E2 29624.469} C_VEL
LIN {X 0,Y 627.132,Z 1052.443,A -85,B 0,C 180,E1 29622.616,E2 29622.616} C_VEL
LIN {X 0,Y 626.09,Z 1067.395,A -85,B 0,C 180,E1 29620.396,E2 29620.396} C_VEL
LIN {X 0,Y 625.343,Z 1079.216,A -85,B 0,C 180,E1 29618.366,E2 29618.366} C_VEL
LIN {X 0,Y 624.799,Z 1089.548,A -85,B 0,C 180,E1 29616.339,E2 29616.339} C_VEL
LIN {X 0,Y 624.377,Z 1099.891,A -85,B 0,C 180,E1 29613.948,E2 29613.948} C_VEL
LIN {X 0,Y 624.15,Z 1107.133,A -85,B 0,C 180,E1 29611.928,E2 29611.928} C_VEL
LIN {X 0,Y 624.023,Z 1112.875,A -85,B 0,C 180,E1 29610,E2 29610} C_VEL
LIN {X 0,Y 623.95,Z 1118.323,A -85,B 0,C 180,E1 29607.704,E2 29607.704} C_VEL
LIN {X 0,Y 623.899,Z 1122.017,A -85,B 0,C 180,E1 29605.404,E2 29605.404} C_VEL
LIN {X 0,Y 623.907,Z 1123.984,A -85,B 0,C 180,E1 29603.467,E2 29603.467} C_VEL
LIN {X 0,Y 623.905,Z 1124.869,A -85,B 0,C 180,E1 29601.522,E2 29601.522} C_VEL
LIN {X 0,Y 623.891,Z 1124.533,A -85,B 0,C 180,E1 29599.193,E2 29599.193} C_VEL
LIN {X 0,Y 623.911,Z 1122.553,A -85,B 0,C 180,E1 29596.941,E2 29596.941} C_VEL
LIN {X 0,Y 623.915,Z 1119.792,A -85,B 0,C 180,E1 29595.048,E2 29595.048} C_VEL
LIN {X 0,Y 623.976,Z 1115.73,A -85,B 0,C 180,E1 29593.044,E2 29593.044} C_VEL
LIN {X 0,Y 624.106,Z 1109.245,A -85,B 0,C 180,E1 29590.632,E2 29590.632} C_VEL
LIN {X 0,Y 624.294,Z 1102.007,A -85,B 0,C 180,E1 29588.521,E2 29588.521} C_VEL
LIN {X 0,Y 624.61,Z 1094.258,A -85,B 0,C 180,E1 29586.61,E2 29586.61} C_VEL
LIN {X 0,Y 625.139,Z 1083.387,A -85,B 0,C 180,E1 29584.314,E2 29584.314} C_VEL
LIN {X 0,Y 625.822,Z 1071.483,A -85,B 0,C 180,E1 29582.191,E2 29582.191} C_VEL
LIN {X 0,Y 626.664,Z 1058.986,A -85,B 0,C 180,E1 29580.227,E2 29580.227} C_VEL
LIN {X 0,Y 627.912,Z 1042.564,A -85,B 0,C 180,E1 29577.977,E2 29577.977} C_VEL
LIN {X 0,Y 629.137,Z 1027.839,A -85,B 0,C 180,E1 29576.204,E2 29576.204} C_VEL
LIN {X 0,Y 630.735,Z 1010.273,A -85,B 0,C 180,E1 29574.313,E2 29574.313} C_VEL
LIN {X 0,Y 632.498,Z 991.04,A -85,B 0,C 180,E1 29572.511,E2 29572.511} C_VEL
LIN {X 0,Y 634.188,Z 973.136,A -85,B 0,C 180,E1 29571.013,E2 29571.013} C_VEL
LIN {X 0,Y 636.311,Z 950.821,A -85,B 0,C 180,E1 29569.375,E2 29569.375} C_VEL
LIN {X 0,Y 638.108,Z 931.326,A -85,B 0,C 180,E1 29568.125,E2 29568.125} C_VEL
LIN {X 0,Y 639.894,Z 911.382,A -85,B 0,C 180,E1 29566.995,E2 29566.995} C_VEL
LIN {X 0,Y 641.956,Z 886.053,A -85,B 0,C 180,E1 29565.765,E2 29565.765} C_VEL
LIN {X 0,Y 643.487,Z 865.378,A -85,B 0,C 180,E1 29564.915,E2 29564.915} C_VEL
LIN {X 0,Y 645.077,Z 842.029,A -85,B 0,C 180,E1 29564.104,E2 29564.104} C_VEL
LIN {X 0,Y 646.592,Z 816.333,A -85,B 0,C 180,E1 29563.391,E2 29563.391} C_VEL
LIN {X 0,Y 647.6,Z 795.464,A -85,B 0,C 180,E1 29562.934,E2 29562.934} C_VEL
LIN {X 0,Y 648.445,Z 771.814,A -85,B 0,C 180,E1 29562.548,E2 29562.548} C_VEL
LIN {X 0,Y 653.194,Z 530.111,A -85,B 0,C 180,E1 29559.367,E2 29559.367} C_VEL
LIN {X 0,Y 656.195,Z 379.264,A -85,B 0,C 180,E1 29557.334,E2 29557.334} C_VEL
LIN {X 0,Y 650.316,Z 353.007,A -85,B 0,C 180,E1 29556.364,E2 29556.364} C_VEL
LIN {X 0,Y 646.321,Z 346.673,A -85,B 0,C 180,E1 29555.843,E2 29555.843} C_VEL
LIN {X 0,Y 639.109,Z 330.487,A -85,B 0,C 180,E1 29553.631,E2 29553.631} C_VEL
LIN {X 0,Y 633.691,Z 319.084,A -85,B 0,C 180,E1 29551.91,E2 29551.91} C_VEL
LIN {X 0,Y 628.895,Z 309.791,A -85,B 0,C 180,E1 29550.371,E2 29550.371} C_VEL
LIN {X 0,Y 626.772,Z 305.545,A -85,B 0,C 180,E1 29549.64,E2 29549.64} C_VEL
LIN {X 0,Y 625,Z 301.809,A -85,B 0,C 180,E1 29548.979,E2 29548.979} C_VEL
LIN {X 0,Y 624.941,Z 301.369,A -85,B 0,C 180,E1 29548.363,E2 29548.363} C_VEL
LIN {X 0,Y 624.944,Z 301.356,A -85,B 0,C 180,E1 29545.087,E2 29545.087} C_VEL
LIN {X 0,Y 624.945,Z 301.35,A -85,B 0,C 180,E1 29541.883,E2 29541.883} C_VEL
LIN {X 0,Y 624.934,Z 301.379,A -85,B 0,C 180,E1 29538.663,E2 29538.663} C_VEL
LIN {X 0,Y 624.939,Z 301.371,A -85,B 0,C 180,E1 29535.498,E2 29535.498} C_VEL
LIN {X 0,Y 624.929,Z 301.35,A -85,B 0,C 180,E1 29532.38,E2 29532.38} C_VEL
LIN {X 0,Y 624.937,Z 301.385,A -85,B 0,C 180,E1 29529.3,E2 29529.3} C_VEL
LIN {X 0,Y 624.93,Z 301.352,A -85,B 0,C 180,E1 29526.154,E2 29526.154} C_VEL
LIN {X 0,Y 624.935,Z 301.372,A -85,B 0,C 180,E1 29523.118,E2 29523.118} C_VEL
LIN {X 0,Y 624.935,Z 301.37,A -85,B 0,C 180,E1 29520,E2 29520} C_VEL
LIN {X 0,Y 624.931,Z 301.354,A -85,B 0,C 180,E1 29516.882,E2 29516.882} C_VEL
LIN {X 0,Y 624.938,Z 301.382,A -85,B 0,C 180,E1 29513.754,E2 29513.754} C_VEL
LIN {X 0,Y 624.928,Z 301.346,A -85,B 0,C 180,E1 29510.7,E2 29510.7} C_VEL
LIN {X 0,Y 624.939,Z 301.388,A -85,B 0,C 180,E1 29507.62,E2 29507.62} C_VEL
LIN {X 0,Y 624.928,Z 301.358,A -85,B 0,C 180,E1 29504.502,E2 29504.502} C_VEL
LIN {X 0,Y 624.94,Z 301.361,A -85,B 0,C 180,E1 29501.434,E2 29501.434} C_VEL
LIN {X 0,Y 624.934,Z 301.387,A -85,B 0,C 180,E1 29498.309,E2 29498.309} C_VEL
LIN {X 0,Y 624.939,Z 301.35,A -85,B 0,C 180,E1 29495.216,E2 29495.216} C_VEL
LIN {X 0,Y 624.928,Z 301.361,A -85,B 0,C 180,E1 29492.147,E2 29492.147} C_VEL
LIN {X 0,Y 624.948,Z 301.385,A -85,B 0,C 180,E1 29488.99,E2 29488.99} C_VEL
LIN {X 0,Y 624.98,Z 301.634,A -85,B 0,C 180,E1 29486.608,E2 29486.608} C_VEL
LIN {X 0,Y 626.407,Z 305.115,A -85,B 0,C 180,E1 29486.035,E2 29486.035} C_VEL
LIN {X 0,Y 627.743,Z 307.064,A -85,B 0,C 180,E1 29485.676,E2 29485.676} C_VEL
LIN {X 0,Y 629.928,Z 310.989,A -85,B 0,C 180,E1 29485.039,E2 29485.039} C_VEL
LIN {X 0,Y 637.247,Z 325.121,A -85,B 0,C 180,E1 29482.949,E2 29482.949} C_VEL
LIN {X 0,Y 645.457,Z 341.916,A -85,B 0,C 180,E1 29480.763,E2 29480.763} C_VEL
LIN {X 0,Y 649.932,Z 350.469,A -85,B 0,C 180,E1 29479.748,E2 29479.748} C_VEL
LIN {X 0,Y 655.978,Z 359.446,A -85,B 0,C 180,E1 29479.04,E2 29479.04} C_VEL
LIN {X 0,Y 661.377,Z 385.116,A -85,B 0,C 180,E1 29478.162,E2 29478.162} C_VEL
LIN {X 0,Y 657.856,Z 583.807,A -85,B 0,C 180,E1 29475.484,E2 29475.484} C_VEL
LIN {X 0,Y 653.636,Z 808.313,A -85,B 0,C 180,E1 29472.492,E2 29472.492} C_VEL
LIN {X 0,Y 652.608,Z 840.695,A -85,B 0,C 180,E1 29472.004,E2 29472.004} C_VEL
LIN {X 0,Y 651.455,Z 864.111,A -85,B 0,C 180,E1 29471.512,E2 29471.512} C_VEL
LIN {X 0,Y 650.123,Z 886.373,A -85,B 0,C 180,E1 29470.921,E2 29470.921} C_VEL
LIN {X 0,Y 648.325,Z 912.629,A -85,B 0,C 180,E1 29470.066,E2 29470.066} C_VEL
LIN {X 0,Y 646.182,Z 938.348,A -85,B 0,C 180,E1 29469.032,E2 29469.032} C_VEL
LIN {X 0,Y 644.374,Z 958.699,A -85,B 0,C 180,E1 29468.082,E2 29468.082} C_VEL
LIN {X 0,Y 642.406,Z 979.36,A -85,B 0,C 180,E1 29466.987,E2 29466.987} C_VEL
LIN {X 0,Y 639.993,Z 1003.726,A -85,B 0,C 180,E1 29465.513,E2 29465.513} C_VEL
LIN {X 0,Y 637.697,Z 1025.638,A -85,B 0,C 180,E1 29463.979,E2 29463.979} C_VEL
LIN {X 0,Y 635.817,Z 1043.509,A -85,B 0,C 180,E1 29462.583,E2 29462.583} C_VEL
LIN {X 0,Y 633.97,Z 1061.274,A -85,B 0,C 180,E1 29461.046,E2 29461.046} C_VEL
LIN {X 0,Y 631.755,Z 1082.667,A -85,B 0,C 180,E1 29458.966,E2 29458.966} C_VEL
LIN {X 0,Y 630.187,Z 1098.845,A -85,B 0,C 180,E1 29457.19,E2 29457.19} C_VEL
LIN {X 0,Y 628.766,Z 1114.165,A -85,B 0,C 180,E1 29455.326,E2 29455.326} C_VEL
LIN {X 0,Y 627.338,Z 1131.251,A -85,B 0,C 180,E1 29452.985,E2 29452.985} C_VEL
LIN {X 0,Y 626.315,Z 1144.86,A -85,B 0,C 180,E1 29450.855,E2 29450.855} C_VEL
LIN {X 0,Y 625.553,Z 1156.307,A -85,B 0,C 180,E1 29448.837,E2 29448.837} C_VEL
LIN {X 0,Y 624.896,Z 1168.202,A -85,B 0,C 180,E1 29446.452,E2 29446.452} C_VEL
LIN {X 0,Y 624.452,Z 1178.088,A -85,B 0,C 180,E1 29444.086,E2 29444.086} C_VEL
LIN {X 0,Y 624.187,Z 1185.798,A -85,B 0,C 180,E1 29441.926,E2 29441.926} C_VEL
LIN {X 0,Y 624.035,Z 1192.621,A -85,B 0,C 180,E1 29439.592,E2 29439.592} C_VEL
LIN {X 0,Y 623.952,Z 1198.251,A -85,B 0,C 180,E1 29437.088,E2 29437.088} C_VEL
LIN {X 0,Y 623.914,Z 1202.013,A -85,B 0,C 180,E1 29434.688,E2 29434.688} C_VEL
LIN {X 0,Y 623.909,Z 1204.208,A -85,B 0,C 180,E1 29432.388,E2 29432.388} C_VEL
LIN {X 0,Y 623.902,Z 1204.961,A -85,B 0,C 180,E1 29429.816,E2 29429.816} C_VEL
LIN {X 0,Y 623.908,Z 1204.072,A -85,B 0,C 180,E1 29427.428,E2 29427.428} C_VEL
LIN {X 0,Y 623.916,Z 1201.899,A -85,B 0,C 180,E1 29425.22,E2 29425.22} C_VEL
LIN {X 0,Y 623.958,Z 1198.079,A -85,B 0,C 180,E1 29422.82,E2 29422.82} C_VEL
LIN {X 0,Y 624.038,Z 1192.377,A -85,B 0,C 180,E1 29420.315,E2 29420.315} C_VEL
LIN {X 0,Y 624.194,Z 1185.494,A -85,B 0,C 180,E1 29417.981,E2 29417.981} C_VEL
LIN {X 0,Y 624.485,Z 1177.372,A -85,B 0,C 180,E1 29415.726,E2 29415.726} C_VEL
LIN {X 0,Y 624.975,Z 1166.375,A -85,B 0,C 180,E1 29413.168,E2 29413.168} C_VEL
LIN {X 0,Y 625.586,Z 1155.797,A -85,B 0,C 180,E1 29411.068,E2 29411.068} C_VEL
LIN {X 0,Y 626.355,Z 1144.275,A -85,B 0,C 180,E1 29409.048,E2 29409.048} C_VEL
LIN {X 0,Y 627.5,Z 1129.3,A -85,B 0,C 180,E1 29406.724,E2 29406.724} C_VEL
LIN {X 0,Y 628.841,Z 1113.386,A -85,B 0,C 180,E1 29404.576,E2 29404.576} C_VEL
LIN {X 0,Y 630.262,Z 1097.999,A -85,B 0,C 180,E1 29402.711,E2 29402.711} C_VEL
LIN {X 0,Y 632.18,Z 1078.815,A -85,B 0,C 180,E1 29400.633,E2 29400.633} C_VEL
LIN {X 0,Y 634.137,Z 1059.613,A -85,B 0,C 180,E1 29398.805,E2 29398.805} C_VEL
LIN {X 0,Y 635.948,Z 1042.23,A -85,B 0,C 180,E1 29397.312,E2 29397.312} C_VEL
LIN {X 0,Y 637.972,Z 1022.963,A -85,B 0,C 180,E1 29395.821,E2 29395.821} C_VEL
LIN {X 0,Y 640.479,Z 998.678,A -85,B 0,C 180,E1 29394.168,E2 29394.168} C_VEL
LIN {X 0,Y 642.579,Z 977.651,A -85,B 0,C 180,E1 29392.918,E2 29392.918} C_VEL
LIN {X 0,Y 644.473,Z 957.702,A -85,B 0,C 180,E1 29391.868,E2 29391.868} C_VEL
LIN {X 0,Y 646.514,Z 934.954,A -85,B 0,C 180,E1 29390.82,E2 29390.82} C_VEL
LIN {X 0,Y 648.636,Z 907.83,A -85,B 0,C 180,E1 29389.769,E2 29389.769} C_VEL
LIN {X 0,Y 650.217,Z 884.868,A -85,B 0,C 180,E1 29389.035,E2 29389.035} C_VEL
LIN {X 0,Y 651.532,Z 862.753,A -85,B 0,C 180,E1 29388.456,E2 29388.456} C_VEL
LIN {X 0,Y 652.799,Z 836.951,A -85,B 0,C 180,E1 29387.926,E2 29387.926} C_VEL
LIN {X 0,Y 653.805,Z 799.113,A -85,B 0,C 180,E1 29387.387,E2 29387.387} C_VEL
LIN {X 0,Y 658.1,Z 571.742,A -85,B 0,C 180,E1 29384.353,E2 29384.353} C_VEL
LIN {X 0,Y 661.396,Z 384.055,A -85,B 0,C 180,E1 29381.813,E2 29381.813} C_VEL
LIN {X 0,Y 655.779,Z 358.723,A -85,B 0,C 180,E1 29380.91,E2 29380.91} C_VEL
LIN {X 0,Y 649.32,Z 349.329,A -85,B 0,C 180,E1 29380.125,E2 29380.125} C_VEL
LIN {X 0,Y 638.697,Z 328.216,A -85,B 0,C 180,E1 29377.468,E2 29377.468} C_VEL
LIN {X 0,Y 631.2,Z 314.104,A -85,B 0,C 180,E1 29375.547,E2 29375.547} C_VEL
LIN {X 0,Y 628.825,Z 309.611,A -85,B 0,C 180,E1 29374.92,E2 29374.92} C_VEL
LIN {X 0,Y 626.871,Z 305.687,A -85,B 0,C 180,E1 29374.378,E2 29374.378} C_VEL
LIN {X 0,Y 625.119,Z 302.381,A -85,B 0,C 180,E1 29373.889,E2 29373.889} C_VEL
LIN {X 0,Y 624.95,Z 301.512,A -85,B 0,C 180,E1 29373.701,E2 29373.701} C_VEL
LIN {X 0,Y 624.941,Z 301.352,A -85,B 0,C 180,E1 29370.584,E2 29370.584} C_VEL
LIN {X 0,Y 624.938,Z 301.349,A -85,B 0,C 180,E1 29367.439,E2 29367.439} C_VEL
LIN {X 0,Y 624.952,Z 301.384,A -85,B 0,C 180,E1 29364.179,E2 29364.179} C_VEL
LIN {X 0,Y 624.94,Z 301.348,A -85,B 0,C 180,E1 29360.904,E2 29360.904} C_VEL
LIN {X 0,Y 624.943,Z 301.376,A -85,B 0,C 180,E1 29357.794,E2 29357.794} C_VEL
LIN {X 0,Y 624.935,Z 301.354,A -85,B 0,C 180,E1 29354.643,E2 29354.643} C_VEL
LIN {X 0,Y 624.941,Z 301.372,A -85,B 0,C 180,E1 29351.537,E2 29351.537} C_VEL
LIN {X 0,Y 624.927,Z 301.353,A -85,B 0,C 180,E1 29348.372,E2 29348.372} C_VEL
LIN {X 0,Y 624.942,Z 301.382,A -85,B 0,C 180,E1 29345.325,E2 29345.325} C_VEL
LIN {X 0,Y 624.928,Z 301.381,A -85,B 0,C 180,E1 29342.201,E2 29342.201} C_VEL
LIN {X 0,Y 624.943,Z 301.385,A -85,B 0,C 180,E1 29339.083,E2 29339.083} C_VEL
LIN {X 0,Y 624.924,Z 301.386,A -85,B 0,C 180,E1 29335.963,E2 29335.963} C_VEL
LIN {X 0,Y 624.946,Z 301.378,A -85,B 0,C 180,E1 29332.831,E2 29332.831} C_VEL
LIN {X 0,Y 624.921,Z 301.382,A -85,B 0,C 180,E1 29329.731,E2 29329.731} C_VEL
LIN {X 0,Y 624.947,Z 301.375,A -85,B 0,C 180,E1 29326.585,E2 29326.585} C_VEL
LIN {X 0,Y 624.918,Z 301.374,A -85,B 0,C 180,E1 29323.548,E2 29323.548} C_VEL
LIN {X 0,Y 624.951,Z 301.378,A -85,B 0,C 180,E1 29320.367,E2 29320.367} C_VEL
LIN {X 0,Y 624.918,Z 301.382,A -85,B 0,C 180,E1 29317.318,E2 29317.318} C_VEL
LIN {X 0,Y 624.943,Z 301.341,A -85,B 0,C 180,E1 29314.1,E2 29314.1} C_VEL
LIN {X 0,Y 624.925,Z 301.383,A -85,B 0,C 180,E1 29311,E2 29311} C_VEL
LIN {X 0,Y 624.92,Z 301.351,A -85,B 0,C 180,E1 29307.696,E2 29307.696} C_VEL
LIN {X 0,Y 624.934,Z 301.376,A -85,B 0,C 180,E1 29304.683,E2 29304.683} C_VEL
LIN {X 0,Y 624.913,Z 301.368,A -85,B 0,C 180,E1 29301.48,E2 29301.48} C_VEL
LIN {X 0,Y 624.93,Z 301.35,A -85,B 0,C 180,E1 29298.484,E2 29298.484} C_VEL
LIN {X 0,Y 624.908,Z 301.386,A -85,B 0,C 180,E1 29295.268,E2 29295.268} C_VEL
LIN {X 0,Y 624.946,Z 301.473,A -85,B 0,C 180,E1 29292.324,E2 29292.324} C_VEL
LIN {X 0,Y 625.066,Z 302.072,A -85,B 0,C 180,E1 29292.164,E2 29292.164} C_VEL
LIN {X 0,Y 626.568,Z 305.296,A -85,B 0,C 180,E1 29291.682,E2 29291.682} C_VEL
LIN {X 0,Y 630.45,Z 313.328,A -85,B 0,C 180,E1 29290.512,E2 29290.512} C_VEL
LIN {X 0,Y 631.09,Z 316.059,A -85,B 0,C 180,E1 29290.196,E2 29290.196} C_VEL
LIN {X 0,Y 630.257,Z 322.986,A -85,B 0,C 180,E1 29289.659,E2 29289.659} C_VEL
LIN {X 0,Y 629.804,Z 328.112,A -85,B 0,C 180,E1 29289.246,E2 29289.246} C_VEL
LIN {X 0,Y 630.36,Z 330.42,A -85,B 0,C 180,E1 29288.981,E2 29288.981} C_VEL
LIN {X 0,Y 638.358,Z 347.456,A -85,B 0,C 180,E1 29286.722,E2 29286.722} C_VEL
LIN {X 0,Y 645.229,Z 358.184,A -85,B 0,C 180,E1 29285.885,E2 29285.885} C_VEL
LIN {X 0,Y 650.512,Z 382.11,A -85,B 0,C 180,E1 29285.014,E2 29285.014} C_VEL
LIN {X 0,Y 645.412,Z 620.697,A -85,B 0,C 180,E1 29281.82,E2 29281.82} C_VEL
LIN {X 0,Y 642.07,Z 781.177,A -85,B 0,C 180,E1 29279.689,E2 29279.689} C_VEL
LIN {X 0,Y 640.933,Z 808.08,A -85,B 0,C 180,E1 29279.183,E2 29279.183} C_VEL
LIN {X 0,Y 639.64,Z 829.862,A -85,B 0,C 180,E1 29278.627,E2 29278.627} C_VEL
LIN {X 0,Y 638.255,Z 849.716,A -85,B 0,C 180,E1 29278.006,E2 29278.006} C_VEL
LIN {X 0,Y 636.564,Z 871.341,A -85,B 0,C 180,E1 29277.199,E2 29277.199} C_VEL
LIN {X 0,Y 634.436,Z 896.469,A -85,B 0,C 180,E1 29276.085,E2 29276.085} C_VEL
LIN {X 0,Y 632.629,Z 916.31,A -85,B 0,C 180,E1 29275.06,E2 29275.06} C_VEL
LIN {X 0,Y 630.696,Z 936.562,A -85,B 0,C 180,E1 29273.87,E2 29273.87} C_VEL
LIN {X 0,Y 628.379,Z 959.642,A -85,B 0,C 180,E1 29272.302,E2 29272.302} C_VEL
LIN {X 0,Y 626.605,Z 977.218,A -85,B 0,C 180,E1 29270.942,E2 29270.942} C_VEL
LIN {X 0,Y 624.746,Z 995.685,A -85,B 0,C 180,E1 29269.347,E2 29269.347} C_VEL
LIN {X 0,Y 622.836,Z 1014.738,A -85,B 0,C 180,E1 29267.469,E2 29267.469} C_VEL
LIN {X 0,Y 621.395,Z 1029.977,A -85,B 0,C 180,E1 29265.779,E2 29265.779} C_VEL
LIN {X 0,Y 619.914,Z 1046.57,A -85,B 0,C 180,E1 29263.715,E2 29263.715} C_VEL
LIN {X 0,Y 618.753,Z 1060.964,A -85,B 0,C 180,E1 29261.653,E2 29261.653} C_VEL
LIN {X 0,Y 617.836,Z 1073.679,A -85,B 0,C 180,E1 29259.595,E2 29259.595} C_VEL
LIN {X 0,Y 617.056,Z 1086.553,A -85,B 0,C 180,E1 29257.167,E2 29257.167} C_VEL
LIN {X 0,Y 616.608,Z 1095.446,A -85,B 0,C 180,E1 29255.21,E2 29255.21} C_VEL
LIN {X 0,Y 616.287,Z 1103.803,A -85,B 0,C 180,E1 29253.069,E2 29253.069} C_VEL
LIN {X 0,Y 616.05,Z 1111.435,A -85,B 0,C 180,E1 29250.651,E2 29250.651} C_VEL
LIN {X 0,Y 615.972,Z 1116.534,A -85,B 0,C 180,E1 29248.605,E2 29248.605} C_VEL
LIN {X 0,Y 615.915,Z 1120.288,A -85,B 0,C 180,E1 29246.65,E2 29246.65} C_VEL
LIN {X 0,Y 615.897,Z 1123.385,A -85,B 0,C 180,E1 29244.317,E2 29244.317} C_VEL
LIN {X 0,Y 615.916,Z 1124.752,A -85,B 0,C 180,E1 29242.01,E2 29242.01} C_VEL
LIN {X 0,Y 615.893,Z 1124.798,A -85,B 0,C 180,E1 29240.091,E2 29240.091} C_VEL
LIN {X 0,Y 615.909,Z 1123.758,A -85,B 0,C 180,E1 29238.102,E2 29238.102} C_VEL
LIN {X 0,Y 615.929,Z 1121.06,A -85,B 0,C 180,E1 29235.715,E2 29235.715} C_VEL
LIN {X 0,Y 615.968,Z 1116.955,A -85,B 0,C 180,E1 29233.497,E2 29233.497} C_VEL
LIN {X 0,Y 616.058,Z 1112.22,A -85,B 0,C 180,E1 29231.55,E2 29231.55} C_VEL
LIN {X 0,Y 616.202,Z 1105.989,A -85,B 0,C 180,E1 29229.483,E2 29229.483} C_VEL
LIN {X 0,Y 616.562,Z 1096.695,A -85,B 0,C 180,E1 29226.994,E2 29226.994} C_VEL
LIN {X 0,Y 617.011,Z 1087.506,A -85,B 0,C 180,E1 29224.943,E2 29224.943} C_VEL
LIN {X 0,Y 617.646,Z 1076.649,A -85,B 0,C 180,E1 29222.838,E2 29222.838} C_VEL
LIN {X 0,Y 618.595,Z 1063.01,A -85,B 0,C 180,E1 29220.57,E2 29220.57} C_VEL
LIN {X 0,Y 619.619,Z 1050.169,A -85,B 0,C 180,E1 29218.695,E2 29218.695} C_VEL
LIN {X 0,Y 621.056,Z 1033.945,A -85,B 0,C 180,E1 29216.592,E2 29216.592} C_VEL
LIN {X 0,Y 622.623,Z 1016.874,A -85,B 0,C 180,E1 29214.668,E2 29214.668} C_VEL
LIN {X 0,Y 624.233,Z 1000.591,A -85,B 0,C 180,E1 29213.026,E2 29213.026} C_VEL
LIN {X 0,Y 626.395,Z 979.438,A -85,B 0,C 180,E1 29211.148,E2 29211.148} C_VEL
LIN {X 0,Y 628.199,Z 961.477,A -85,B 0,C 180,E1 29209.744,E2 29209.744} C_VEL
LIN {X 0,Y 630.319,Z 940.464,A -85,B 0,C 180,E1 29208.284,E2 29208.284} C_VEL
LIN {X 0,Y 632.493,Z 917.739,A -85,B 0,C 180,E1 29206.928,E2 29206.928} C_VEL
LIN {X 0,Y 634.191,Z 899.031,A -85,B 0,C 180,E1 29205.951,E2 29205.951} C_VEL
LIN {X 0,Y 636.249,Z 875.491,A -85,B 0,C 180,E1 29204.88,E2 29204.88} C_VEL
LIN {X 0,Y 638.184,Z 851.295,A -85,B 0,C 180,E1 29203.954,E2 29203.954} C_VEL
LIN {X 0,Y 639.619,Z 830.923,A -85,B 0,C 180,E1 29203.308,E2 29203.308} C_VEL
LIN {X 0,Y 640.847,Z 810.522,A -85,B 0,C 180,E1 29202.779,E2 29202.779} C_VEL
LIN {X 0,Y 642.046,Z 785.089,A -85,B 0,C 180,E1 29202.274,E2 29202.274} C_VEL
LIN {X 0,Y 643.218,Z 734.571,A -85,B 0,C 180,E1 29201.582,E2 29201.582} C_VEL
LIN {X 0,Y 648.258,Z 494.974,A -85,B 0,C 180,E1 29198.398,E2 29198.398} C_VEL
LIN {X 0,Y 650.618,Z 381.175,A -85,B 0,C 180,E1 29196.845,E2 29196.845} C_VEL
LIN {X 0,Y 645.484,Z 357.861,A -85,B 0,C 180,E1 29195.965,E2 29195.965} C_VEL
LIN {X 0,Y 638.189,Z 346.574,A -85,B 0,C 180,E1 29194.99,E2 29194.99} C_VEL
LIN {X 0,Y 630.495,Z 329.386,A -85,B 0,C 180,E1 29192.522,E2 29192.522} C_VEL
LIN {X 0,Y 625.376,Z 319.302,A -85,B 0,C 180,E1 29190.88,E2 29190.88} C_VEL
LIN {X 0,Y 623.473,Z 315.498,A -85,B 0,C 180,E1 29190.237,E2 29190.237} C_VEL
LIN {X 0,Y 621.113,Z 310.956,A -85,B 0,C 180,E1 29189.437,E2 29189.437} C_VEL
LIN {X 0,Y 618.952,Z 306.703,A -85,B 0,C 180,E1 29188.672,E2 29188.672} C_VEL
LIN {X 0,Y 617.142,Z 303.127,A -85,B 0,C 180,E1 29187.996,E2 29187.996} C_VEL
LIN {X 0,Y 617.014,Z 302.459,A -85,B 0,C 180,E1 29187.775,E2 29187.775} C_VEL
LIN {X 0,Y 616.99,Z 302.352,A -85,B 0,C 180,E1 29184.716,E2 29184.716} C_VEL
LIN {X 0,Y 616.999,Z 302.336,A -85,B 0,C 180,E1 29181.684,E2 29181.684} C_VEL
LIN {X 0,Y 616.993,Z 302.36,A -85,B 0,C 180,E1 29178.52,E2 29178.52} C_VEL
LIN {X 0,Y 616.999,Z 302.363,A -85,B 0,C 180,E1 29175.376,E2 29175.376} C_VEL
LIN {X 0,Y 616.99,Z 302.336,A -85,B 0,C 180,E1 29172.257,E2 29172.257} C_VEL
LIN {X 0,Y 616.999,Z 302.372,A -85,B 0,C 180,E1 29169.138,E2 29169.138} C_VEL
LIN {X 0,Y 616.995,Z 302.342,A -85,B 0,C 180,E1 29165.953,E2 29165.953} C_VEL
LIN {X 0,Y 617.003,Z 302.353,A -85,B 0,C 180,E1 29162.787,E2 29162.787} C_VEL
LIN {X 0,Y 617.014,Z 302.364,A -85,B 0,C 180,E1 29159.536,E2 29159.536} C_VEL
LIN {X 0,Y 617.003,Z 302.332,A -85,B 0,C 180,E1 29156.283,E2 29156.283} C_VEL
LIN {X 0,Y 617.004,Z 302.374,A -85,B 0,C 180,E1 29153.112,E2 29153.112} C_VEL
LIN {X 0,Y 617,Z 302.337,A -85,B 0,C 180,E1 29149.92,E2 29149.92} C_VEL
LIN {X 0,Y 616.993,Z 302.358,A -85,B 0,C 180,E1 29146.791,E2 29146.791} C_VEL
LIN {X 0,Y 617.002,Z 302.363,A -85,B 0,C 180,E1 29143.718,E2 29143.718} C_VEL
LIN {X 0,Y 616.988,Z 302.336,A -85,B 0,C 180,E1 29140.589,E2 29140.589} C_VEL
LIN {X 0,Y 617.005,Z 302.371,A -85,B 0,C 180,E1 29137.471,E2 29137.471} C_VEL
LIN {X 0,Y 616.989,Z 302.354,A -85,B 0,C 180,E1 29134.361,E2 29134.361} C_VEL
LIN {X 0,Y 617,Z 302.336,A -85,B 0,C 180,E1 29131.229,E2 29131.229} C_VEL
LIN {X 0,Y 616.989,Z 302.369,A -85,B 0,C 180,E1 29128.217,E2 29128.217} C_VEL
LIN {X 0,Y 617.082,Z 302.828,A -85,B 0,C 180,E1 29127.597,E2 29127.597} C_VEL
LIN {X 0,Y 618.654,Z 306.326,A -85,B 0,C 180,E1 29126.998,E2 29126.998} C_VEL
LIN {X 0,Y 619.914,Z 308.277,A -85,B 0,C 180,E1 29126.632,E2 29126.632} C_VEL
LIN {X 0,Y 622.037,Z 312.03,A -85,B 0,C 180,E1 29125.986,E2 29125.986} C_VEL
LIN {X 0,Y 627.864,Z 323.087,A -85,B 0,C 180,E1 29124.235,E2 29124.235} C_VEL
LIN {X 0,Y 634.3,Z 335.873,A -85,B 0,C 180,E1 29122.406,E2 29122.406} C_VEL
LIN {X 0,Y 641.356,Z 350.231,A -85,B 0,C 180,E1 29120.586,E2 29120.586} C_VEL
LIN {X 0,Y 650.939,Z 364.046,A -85,B 0,C 180,E1 29119.433,E2 29119.433} C_VEL
LIN {X 0,Y 655.713,Z 386.987,A -85,B 0,C 180,E1 29118.635,E2 29118.635} C_VEL
LIN {X 0,Y 651.854,Z 599.381,A -85,B 0,C 180,E1 29115.771,E2 29115.771} C_VEL
LIN {X 0,Y 647.503,Z 818.376,A -85,B 0,C 180,E1 29112.835,E2 29112.835} C_VEL
LIN {X 0,Y 646.518,Z 843.413,A -85,B 0,C 180,E1 29112.429,E2 29112.429} C_VEL
LIN {X 0,Y 645.348,Z 865.541,A -85,B 0,C 180,E1 29111.952,E2 29111.952} C_VEL
LIN {X 0,Y 643.874,Z 888.634,A -85,B 0,C 180,E1 29111.327,E2 29111.327} C_VEL
LIN {X 0,Y 641.709,Z 917.057,A -85,B 0,C 180,E1 29110.364,E2 29110.364} C_VEL
LIN {X 0,Y 639.768,Z 939.128,A -85,B 0,C 180,E1 29109.459,E2 29109.459} C_VEL
LIN {X 0,Y 637.82,Z 959.701,A -85,B 0,C 180,E1 29108.488,E2 29108.488} C_VEL
LIN {X 0,Y 635.632,Z 981.248,A -85,B 0,C 180,E1 29107.329,E2 29107.329} C_VEL
LIN {X 0,Y 632.926,Z 1006.39,A -85,B 0,C 180,E1 29105.768,E2 29105.768} C_VEL
LIN {X 0,Y 630.712,Z 1026.236,A -85,B 0,C 180,E1 29104.358,E2 29104.358} C_VEL
LIN {X 0,Y 628.712,Z 1044.055,A -85,B 0,C 180,E1 29102.949,E2 29102.949} C_VEL
LIN {X 0,Y 626.562,Z 1063.489,A -85,B 0,C 180,E1 29101.24,E2 29101.24} C_VEL
LIN {X 0,Y 624.266,Z 1083.988,A -85,B 0,C 180,E1 29099.199,E2 29099.199} C_VEL
LIN {X 0,Y 622.629,Z 1099.688,A -85,B 0,C 180,E1 29097.444,E2 29097.444} C_VEL
LIN {X 0,Y 621.012,Z 1116.092,A -85,B 0,C 180,E1 29095.409,E2 29095.409} C_VEL
LIN {X 0,Y 619.468,Z 1133.187,A -85,B 0,C 180,E1 29092.992,E2 29092.992} C_VEL
LIN {X 0,Y 618.445,Z 1146.008,A -85,B 0,C 180,E1 29090.934,E2 29090.934} C_VEL
LIN {X 0,Y 617.578,Z 1158.364,A -85,B 0,C 180,E1 29088.697,E2 29088.697} C_VEL
LIN {X 0,Y 616.881,Z 1170.261,A -85,B 0,C 180,E1 29086.188,E2 29086.188} C_VEL
LIN {X 0,Y 616.475,Z 1178.804,A -85,B 0,C 180,E1 29084.081,E2 29084.081} C_VEL
LIN {X 0,Y 616.204,Z 1186.098,A -85,B 0,C 180,E1 29081.987,E2 29081.987} C_VEL
LIN {X 0,Y 616.039,Z 1193.108,A -85,B 0,C 180,E1 29079.529,E2 29079.529} C_VEL
LIN {X 0,Y 615.947,Z 1198.594,A -85,B 0,C 180,E1 29076.993,E2 29076.993} C_VEL
LIN {X 0,Y 615.914,Z 1202.124,A -85,B 0,C 180,E1 29074.656,E2 29074.656} C_VEL
LIN {X 0,Y 615.911,Z 1204.27,A -85,B 0,C 180,E1 29072.326,E2 29072.326} C_VEL
LIN {X 0,Y 615.897,Z 1204.939,A -85,B 0,C 180,E1 29069.721,E2 29069.721} C_VEL
LIN {X 0,Y 615.908,Z 1204.069,A -85,B 0,C 180,E1 29067.395,E2 29067.395} C_VEL
LIN {X 0,Y 615.918,Z 1201.896,A -85,B 0,C 180,E1 29065.158,E2 29065.158} C_VEL
LIN {X 0,Y 615.961,Z 1197.989,A -85,B 0,C 180,E1 29062.677,E2 29062.677} C_VEL
LIN {X 0,Y 616.053,Z 1192.224,A -85,B 0,C 180,E1 29060.131,E2 29060.131} C_VEL
LIN {X 0,Y 616.22,Z 1185.491,A -85,B 0,C 180,E1 29057.823,E2 29057.823} C_VEL
LIN {X 0,Y 616.551,Z 1177.267,A -85,B 0,C 180,E1 29055.509,E2 29055.509} C_VEL
LIN {X 0,Y 617.081,Z 1166.36,A -85,B 0,C 180,E1 29052.943,E2 29052.943} C_VEL
LIN {X 0,Y 617.736,Z 1155.795,A -85,B 0,C 180,E1 29050.818,E2 29050.818} C_VEL
LIN {X 0,Y 618.572,Z 1144.284,A -85,B 0,C 180,E1 29048.773,E2 29048.773} C_VEL
LIN {X 0,Y 619.831,Z 1129.089,A -85,B 0,C 180,E1 29046.389,E2 29046.389} C_VEL
LIN {X 0,Y 621.28,Z 1113.393,A -85,B 0,C 180,E1 29044.245,E2 29044.245} C_VEL
LIN {X 0,Y 622.789,Z 1097.999,A -85,B 0,C 180,E1 29042.356,E2 29042.356} C_VEL
LIN {X 0,Y 624.875,Z 1078.882,A -85,B 0,C 180,E1 29040.262,E2 29040.262} C_VEL
LIN {X 0,Y 626.91,Z 1060.167,A -85,B 0,C 180,E1 29038.458,E2 29038.458} C_VEL
LIN {X 0,Y 628.843,Z 1042.837,A -85,B 0,C 180,E1 29036.95,E2 29036.95} C_VEL
LIN {X 0,Y 630.916,Z 1024.336,A -85,B 0,C 180,E1 29035.499,E2 29035.499} C_VEL
LIN {X 0,Y 633.601,Z 1000.286,A -85,B 0,C 180,E1 29033.829,E2 29033.829} C_VEL
LIN {X 0,Y 635.914,Z 978.548,A -85,B 0,C 180,E1 29032.52,E2 29032.52} C_VEL
LIN {X 0,Y 637.938,Z 958.562,A -85,B 0,C 180,E1 29031.456,E2 29031.456} C_VEL
LIN {X 0,Y 639.962,Z 937.212,A -85,B 0,C 180,E1 29030.457,E2 29030.457} C_VEL
LIN {X 0,Y 642.287,Z 910.04,A -85,B 0,C 180,E1 29029.376,E2 29029.376} C_VEL
LIN {X 0,Y 644.068,Z 885.644,A -85,B 0,C 180,E1 29028.586,E2 29028.586} C_VEL
LIN {X 0,Y 645.45,Z 863.787,A -85,B 0,C 180,E1 29028.006,E2 29028.006} C_VEL
LIN {X 0,Y 646.658,Z 840.518,A -85,B 0,C 180,E1 29027.516,E2 29027.516} C_VEL
LIN {X 0,Y 647.768,Z 806.8,A -85,B 0,C 180,E1 29027.008,E2 29027.008} C_VEL
LIN {X 0,Y 652.091,Z 586.507,A -85,B 0,C 180,E1 29024.058,E2 29024.058} C_VEL
LIN {X 0,Y 655.811,Z 386.24,A -85,B 0,C 180,E1 29021.343,E2 29021.343} C_VEL
LIN {X 0,Y 650.801,Z 363.519,A -85,B 0,C 180,E1 29020.52,E2 29020.52} C_VEL
LIN {X 0,Y 640.901,Z 349.383,A -85,B 0,C 180,E1 29019.303,E2 29019.303} C_VEL
LIN {X 0,Y 632.68,Z 332.927,A -85,B 0,C 180,E1 29017.203,E2 29017.203} C_VEL
LIN {X 0,Y 625.929,Z 320.018,A -85,B 0,C 180,E1 29015.442,E2 29015.442} C_VEL
LIN {X 0,Y 621.237,Z 311.094,A -85,B 0,C 180,E1 29014.175,E2 29014.175} C_VEL
LIN {X 0,Y 618.567,Z 306.216,A -85,B 0,C 180,E1 29013.451,E2 29013.451} C_VEL
LIN {X 0,Y 617.031,Z 302.573,A -85,B 0,C 180,E1 29012.909,E2 29012.909} C_VEL
LIN {X 0,Y 616.993,Z 302.359,A -85,B 0,C 180,E1 29009.89,E2 29009.89} C_VEL
LIN {X 0,Y 616.996,Z 302.331,A -85,B 0,C 180,E1 29006.777,E2 29006.777} C_VEL
LIN {X 0,Y 616.996,Z 302.371,A -85,B 0,C 180,E1 29003.697,E2 29003.697} C_VEL
LIN {X 0,Y 616.994,Z 302.342,A -85,B 0,C 180,E1 29000.589,E2 29000.589} C_VEL
LIN {X 0,Y 616.996,Z 302.35,A -85,B 0,C 180,E1 28997.446,E2 28997.446} C_VEL
LIN {X 0,Y 616.993,Z 302.353,A -85,B 0,C 180,E1 28994.286,E2 28994.286} C_VEL
LIN {X 0,Y 617.001,Z 302.345,A -85,B 0,C 180,E1 28991.119,E2 28991.119} C_VEL
LIN {X 0,Y 617.001,Z 302.353,A -85,B 0,C 180,E1 28987.918,E2 28987.918} C_VEL
LIN {X 0,Y 617.005,Z 302.364,A -85,B 0,C 180,E1 28984.648,E2 28984.648} C_VEL
LIN {X 0,Y 617.009,Z 302.364,A -85,B 0,C 180,E1 28981.393,E2 28981.393} C_VEL
LIN {X 0,Y 616.99,Z 302.365,A -85,B 0,C 180,E1 28978.236,E2 28978.236} C_VEL
LIN {X 0,Y 617.007,Z 302.373,A -85,B 0,C 180,E1 28975.073,E2 28975.073} C_VEL
LIN {X 0,Y 616.984,Z 302.374,A -85,B 0,C 180,E1 28971.955,E2 28971.955} C_VEL
LIN {X 0,Y 617.008,Z 302.371,A -85,B 0,C 180,E1 28968.786,E2 28968.786} C_VEL
LIN {X 0,Y 616.98,Z 302.374,A -85,B 0,C 180,E1 28965.643,E2 28965.643} C_VEL
LIN {X 0,Y 617.012,Z 302.364,A -85,B 0,C 180,E1 28962.457,E2 28962.457} C_VEL
LIN {X 0,Y 616.985,Z 302.367,A -85,B 0,C 180,E1 28959.311,E2 28959.311} C_VEL
LIN {X 0,Y 617.002,Z 302.341,A -85,B 0,C 180,E1 28956.1,E2 28956.1} C_VEL
LIN {X 0,Y 616.997,Z 302.361,A -85,B 0,C 180,E1 28952.91,E2 28952.91} C_VEL
LIN {X 0,Y 616.982,Z 302.344,A -85,B 0,C 180,E1 28949.734,E2 28949.734} C_VEL
LIN {X 0,Y 617.001,Z 302.364,A -85,B 0,C 180,E1 28946.676,E2 28946.676} C_VEL
LIN {X 0,Y 616.972,Z 302.333,A -85,B 0,C 180,E1 28943.495,E2 28943.495} C_VEL
LIN {X 0,Y 617.011,Z 302.374,A -85,B 0,C 180,E1 28940.441,E2 28940.441} C_VEL
LIN {X 0,Y 616.964,Z 302.341,A -85,B 0,C 180,E1 28937.23,E2 28937.23} C_VEL
LIN {X 0,Y 617.004,Z 302.336,A -85,B 0,C 180,E1 28934.251,E2 28934.251} C_VEL
LIN {X 0,Y 616.996,Z 302.603,A -85,B 0,C 180,E1 28933.084,E2 28933.084} C_VEL
LIN {X 0,Y 618.556,Z 306.232,A -85,B 0,C 180,E1 28932.513,E2 28932.513} C_VEL
LIN {X 0,Y 621.917,Z 313.118,A -85,B 0,C 180,E1 28931.477,E2 28931.477} C_VEL
LIN {X 0,Y 627.689,Z 324.782,A -85,B 0,C 180,E1 28929.771,E2 28929.771} C_VEL
LIN {X 0,Y 630.36,Z 330.42,A -85,B 0,C 180,E1 28928.981,E2 28928.981} C_VEL
LIN {X 0,Y 631.275,Z 334.229,A -85,B 0,C 180,E1 28928.558,E2 28928.558} C_VEL
LIN {X 0,Y 630.65,Z 340.543,A -85,B 0,C 180,E1 28928.056,E2 28928.056} C_VEL
LIN {X 0,Y 630.037,Z 346.951,A -85,B 0,C 180,E1 28927.579,E2 28927.579} C_VEL
LIN {X 0,Y 630.453,Z 347.987,A -85,B 0,C 180,E1 28927.494,E2 28927.494} C_VEL
LIN {X 0,Y 640.257,Z 362.758,A -85,B 0,C 180,E1 28926.286,E2 28926.286} C_VEL
LIN {X 0,Y 644.948,Z 384.292,A -85,B 0,C 180,E1 28925.502,E2 28925.502} C_VEL
LIN {X 0,Y 639.57,Z 622.062,A -85,B 0,C 180,E1 28922.296,E2 28922.296} C_VEL
LIN {X 0,Y 636.049,Z 781.543,A -85,B 0,C 180,E1 28920.162,E2 28920.162} C_VEL
LIN {X 0,Y 634.86,Z 808.353,A -85,B 0,C 180,E1 28919.655,E2 28919.655} C_VEL
LIN {X 0,Y 633.481,Z 830.469,A -85,B 0,C 180,E1 28919.087,E2 28919.087} C_VEL
LIN {X 0,Y 632.021,Z 850.313,A -85,B 0,C 180,E1 28918.462,E2 28918.462} C_VEL
LIN {X 0,Y 630.235,Z 871.918,A -85,B 0,C 180,E1 28917.648,E2 28917.648} C_VEL
LIN {X 0,Y 627.893,Z 896.55,A -85,B 0,C 180,E1 28916.53,E2 28916.53} C_VEL
LIN {X 0,Y 625.722,Z 917.671,A -85,B 0,C 180,E1 28915.407,E2 28915.407} C_VEL
LIN {X 0,Y 623.405,Z 940.397,A -85,B 0,C 180,E1 28914.04,E2 28914.04} C_VEL
LIN {X 0,Y 621.142,Z 961.284,A -85,B 0,C 180,E1 28912.576,E2 28912.576} C_VEL
LIN {X 0,Y 619.213,Z 979.295,A -85,B 0,C 180,E1 28911.155,E2 28911.155} C_VEL
LIN {X 0,Y 616.964,Z 999.994,A -85,B 0,C 180,E1 28909.305,E2 28909.305} C_VEL
LIN {X 0,Y 615.181,Z 1016.773,A -85,B 0,C 180,E1 28907.596,E2 28907.596} C_VEL
LIN {X 0,Y 613.599,Z 1032.645,A -85,B 0,C 180,E1 28905.791,E2 28905.791} C_VEL
LIN {X 0,Y 611.977,Z 1049.488,A -85,B 0,C 180,E1 28903.607,E2 28903.607} C_VEL
LIN {X 0,Y 610.882,Z 1062.372,A -85,B 0,C 180,E1 28901.71,E2 28901.71} C_VEL
LIN {X 0,Y 609.854,Z 1075.997,A -85,B 0,C 180,E1 28899.436,E2 28899.436} C_VEL
LIN {X 0,Y 609.123,Z 1087.129,A -85,B 0,C 180,E1 28897.261,E2 28897.261} C_VEL
LIN {X 0,Y 608.65,Z 1095.953,A -85,B 0,C 180,E1 28895.278,E2 28895.278} C_VEL
LIN {X 0,Y 608.294,Z 1104.906,A -85,B 0,C 180,E1 28892.921,E2 28892.921} C_VEL
LIN {X 0,Y 608.057,Z 1111.756,A -85,B 0,C 180,E1 28890.659,E2 28890.659} C_VEL
LIN {X 0,Y 607.978,Z 1116.589,A -85,B 0,C 180,E1 28888.681,E2 28888.681} C_VEL
LIN {X 0,Y 607.919,Z 1120.33,A -85,B 0,C 180,E1 28886.7,E2 28886.7} C_VEL
LIN {X 0,Y 607.897,Z 1123.471,A -85,B 0,C 180,E1 28884.242,E2 28884.242} C_VEL
LIN {X 0,Y 607.917,Z 1124.743,A -85,B 0,C 180,E1 28882.059,E2 28882.059} C_VEL
LIN {X 0,Y 607.894,Z 1124.792,A -85,B 0,C 180,E1 28880.055,E2 28880.055} C_VEL
LIN {X 0,Y 607.909,Z 1123.67,A -85,B 0,C 180,E1 28877.943,E2 28877.943} C_VEL
LIN {X 0,Y 607.924,Z 1120.69,A -85,B 0,C 180,E1 28875.425,E2 28875.425} C_VEL
LIN {X 0,Y 607.983,Z 1116.684,A -85,B 0,C 180,E1 28873.274,E2 28873.274} C_VEL
LIN {X 0,Y 608.077,Z 1111.858,A -85,B 0,C 180,E1 28871.289,E2 28871.289} C_VEL
LIN {X 0,Y 608.3,Z 1104.616,A -85,B 0,C 180,E1 28868.902,E2 28868.902} C_VEL
LIN {X 0,Y 608.674,Z 1095.718,A -85,B 0,C 180,E1 28866.576,E2 28866.576} C_VEL
LIN {X 0,Y 609.143,Z 1087.05,A -85,B 0,C 180,E1 28864.633,E2 28864.633} C_VEL
LIN {X 0,Y 609.907,Z 1075.376,A -85,B 0,C 180,E1 28862.358,E2 28862.358} C_VEL
LIN {X 0,Y 610.899,Z 1062.123,A -85,B 0,C 180,E1 28860.162,E2 28860.162} C_VEL
LIN {X 0,Y 612.012,Z 1049.183,A -85,B 0,C 180,E1 28858.26,E2 28858.26} C_VEL
LIN {X 0,Y 613.667,Z 1031.836,A -85,B 0,C 180,E1 28856.023,E2 28856.023} C_VEL
LIN {X 0,Y 615.233,Z 1016.179,A -85,B 0,C 180,E1 28854.25,E2 28854.25} C_VEL
LIN {X 0,Y 617.13,Z 998.601,A -85,B 0,C 180,E1 28852.469,E2 28852.469} C_VEL
LIN {X 0,Y 619.239,Z 979.028,A -85,B 0,C 180,E1 28850.732,E2 28850.732} C_VEL
LIN {X 0,Y 621.188,Z 960.847,A -85,B 0,C 180,E1 28849.301,E2 28849.301} C_VEL
LIN {X 0,Y 623.543,Z 939.153,A -85,B 0,C 180,E1 28847.788,E2 28847.788} C_VEL
LIN {X 0,Y 625.884,Z 916.294,A -85,B 0,C 180,E1 28846.423,E2 28846.423} C_VEL
LIN {X 0,Y 628.347,Z 892.589,A -85,B 0,C 180,E1 28845.177,E2 28845.177} C_VEL
LIN {X 0,Y 630.553,Z 868.557,A -85,B 0,C 180,E1 28844.118,E2 28844.118} C_VEL
LIN {X 0,Y 632.274,Z 847.985,A -85,B 0,C 180,E1 28843.358,E2 28843.358} C_VEL
LIN {X 0,Y 634.085,Z 823.073,A -85,B 0,C 180,E1 28842.6,E2 28842.6} C_VEL
LIN {X 0,Y 635.426,Z 798.514,A -85,B 0,C 180,E1 28842.038,E2 28842.038} C_VEL
LIN {X 0,Y 636.335,Z 776.404,A -85,B 0,C 180,E1 28841.66,E2 28841.66} C_VEL
LIN {X 0,Y 641.635,Z 539.069,A -85,B 0,C 180,E1 28838.482,E2 28838.482} C_VEL
LIN {X 0,Y 645.178,Z 383.273,A -85,B 0,C 180,E1 28836.349,E2 28836.349} C_VEL
LIN {X 0,Y 640.687,Z 362.679,A -85,B 0,C 180,E1 28835.559,E2 28835.559} C_VEL
LIN {X 0,Y 630.845,Z 347.865,A -85,B 0,C 180,E1 28834.241,E2 28834.241} C_VEL
LIN {X 0,Y 629.091,Z 344.284,A -85,B 0,C 180,E1 28833.774,E2 28833.774} C_VEL
LIN {X 0,Y 622.761,Z 330.468,A -85,B 0,C 180,E1 28831.67,E2 28831.67} C_VEL
LIN {X 0,Y 616.261,Z 317.431,A -85,B 0,C 180,E1 28829.447,E2 28829.447} C_VEL
LIN {X 0,Y 613.264,Z 312.049,A -85,B 0,C 180,E1 28828.43,E2 28828.43} C_VEL
LIN {X 0,Y 610.98,Z 307.638,A -85,B 0,C 180,E1 28827.59,E2 28827.59} C_VEL
LIN {X 0,Y 609.257,Z 304.385,A -85,B 0,C 180,E1 28826.934,E2 28826.934} C_VEL
LIN {X 0,Y 609.076,Z 303.521,A -85,B 0,C 180,E1 28826.732,E2 28826.732} C_VEL
LIN {X 0,Y 609.066,Z 303.366,A -85,B 0,C 180,E1 28823.717,E2 28823.717} C_VEL
LIN {X 0,Y 609.052,Z 303.336,A -85,B 0,C 180,E1 28820.569,E2 28820.569} C_VEL
LIN {X 0,Y 609.058,Z 303.323,A -85,B 0,C 180,E1 28817.484,E2 28817.484} C_VEL
LIN {X 0,Y 609.057,Z 303.366,A -85,B 0,C 180,E1 28814.353,E2 28814.353} C_VEL
LIN {X 0,Y 609.058,Z 303.331,A -85,B 0,C 180,E1 28811.17,E2 28811.17} C_VEL
LIN {X 0,Y 609.056,Z 303.333,A -85,B 0,C 180,E1 28808.022,E2 28808.022} C_VEL
LIN {X 0,Y 609.067,Z 303.361,A -85,B 0,C 180,E1 28804.803,E2 28804.803} C_VEL
LIN {X 0,Y 609.065,Z 303.32,A -85,B 0,C 180,E1 28801.505,E2 28801.505} C_VEL
LIN {X 0,Y 609.07,Z 303.361,A -85,B 0,C 180,E1 28798.307,E2 28798.307} C_VEL
LIN {X 0,Y 609.058,Z 303.328,A -85,B 0,C 180,E1 28795.103,E2 28795.103} C_VEL
LIN {X 0,Y 609.061,Z 303.34,A -85,B 0,C 180,E1 28791.979,E2 28791.979} C_VEL
LIN {X 0,Y 609.055,Z 303.351,A -85,B 0,C 180,E1 28788.83,E2 28788.83} C_VEL
LIN {X 0,Y 609.058,Z 303.323,A -85,B 0,C 180,E1 28785.647,E2 28785.647} C_VEL
LIN {X 0,Y 609.054,Z 303.362,A -85,B 0,C 180,E1 28782.516,E2 28782.516} C_VEL
LIN {X 0,Y 609.061,Z 303.331,A -85,B 0,C 180,E1 28779.331,E2 28779.331} C_VEL
LIN {X 0,Y 609.049,Z 303.329,A -85,B 0,C 180,E1 28776.283,E2 28776.283} C_VEL
LIN {X 0,Y 609.071,Z 303.359,A -85,B 0,C 180,E1 28773.049,E2 28773.049} C_VEL
LIN {X 0,Y 609.064,Z 303.345,A -85,B 0,C 180,E1 28769.844,E2 28769.844} C_VEL
LIN {X 0,Y 609.115,Z 303.635,A -85,B 0,C 180,E1 28768.753,E2 28768.753} C_VEL
LIN {X 0,Y 610.396,Z 306.901,A -85,B 0,C 180,E1 28768.165,E2 28768.165} C_VEL
LIN {X 0,Y 611.977,Z 309.069,A -85,B 0,C 180,E1 28767.705,E2 28767.705} C_VEL
LIN {X 0,Y 613.949,Z 312.796,A -85,B 0,C 180,E1 28767.046,E2 28767.046} C_VEL
LIN {X 0,Y 617.797,Z 319.891,A -85,B 0,C 180,E1 28765.832,E2 28765.832} C_VEL
LIN {X 0,Y 623.022,Z 329.764,A -85,B 0,C 180,E1 28764.254,E2 28764.254} C_VEL
LIN {X 0,Y 630.202,Z 344.141,A -85,B 0,C 180,E1 28762.196,E2 28762.196} C_VEL
LIN {X 0,Y 633.218,Z 350.384,A -85,B 0,C 180,E1 28761.425,E2 28761.425} C_VEL
LIN {X 0,Y 645.966,Z 368.727,A -85,B 0,C 180,E1 28759.828,E2 28759.828} C_VEL
LIN {X 0,Y 650.102,Z 389.034,A -85,B 0,C 180,E1 28759.115,E2 28759.115} C_VEL
LIN {X 0,Y 645.938,Z 601.275,A -85,B 0,C 180,E1 28756.228,E2 28756.228} C_VEL
LIN {X 0,Y 642.594,Z 773.643,A -85,B 0,C 180,E1 28753.925,E2 28753.925} C_VEL
LIN {X 0,Y 641.207,Z 830.472,A -85,B 0,C 180,E1 28753.142,E2 28753.142} C_VEL
LIN {X 0,Y 639.766,Z 859.313,A -85,B 0,C 180,E1 28752.584,E2 28752.584} C_VEL
LIN {X 0,Y 638.241,Z 882.543,A -85,B 0,C 180,E1 28751.985,E2 28751.985} C_VEL
LIN {X 0,Y 636.65,Z 903.38,A -85,B 0,C 180,E1 28751.33,E2 28751.33} C_VEL
LIN {X 0,Y 634.89,Z 923.87,A -85,B 0,C 180,E1 28750.573,E2 28750.573} C_VEL
LIN {X 0,Y 632.62,Z 948.06,A -85,B 0,C 180,E1 28749.528,E2 28749.528} C_VEL
LIN {X 0,Y 629.981,Z 973.14,A -85,B 0,C 180,E1 28748.242,E2 28748.242} C_VEL
LIN {X 0,Y 627.839,Z 992.195,A -85,B 0,C 180,E1 28747.126,E2 28747.126} C_VEL
LIN {X 0,Y 625.618,Z 1011.292,A -85,B 0,C 180,E1 28745.873,E2 28745.873} C_VEL
LIN {X 0,Y 623.341,Z 1030.544,A -85,B 0,C 180,E1 28744.462,E2 28744.462} C_VEL
LIN {X 0,Y 620.564,Z 1053.505,A -85,B 0,C 180,E1 28742.557,E2 28742.557} C_VEL
LIN {X 0,Y 618.357,Z 1071.784,A -85,B 0,C 180,E1 28740.836,E2 28740.836} C_VEL
LIN {X 0,Y 616.514,Z 1087.768,A -85,B 0,C 180,E1 28739.167,E2 28739.167} C_VEL
LIN {X 0,Y 614.576,Z 1105.603,A -85,B 0,C 180,E1 28737.099,E2 28737.099} C_VEL
LIN {X 0,Y 612.8,Z 1122.414,A -85,B 0,C 180,E1 28734.877,E2 28734.877} C_VEL
LIN {X 0,Y 611.534,Z 1135.74,A -85,B 0,C 180,E1 28732.9,E2 28732.9} C_VEL
LIN {X 0,Y 610.396,Z 1149.445,A -85,B 0,C 180,E1 28730.621,E2 28730.621} C_VEL
LIN {X 0,Y 609.431,Z 1162.687,A -85,B 0,C 180,E1 28728.064,E2 28728.064} C_VEL
LIN {X 0,Y 608.873,Z 1171.901,A -85,B 0,C 180,E1 28726.015,E2 28726.015} C_VEL
LIN {X 0,Y 608.483,Z 1179.868,A -85,B 0,C 180,E1 28723.978,E2 28723.978} C_VEL
LIN {X 0,Y 608.199,Z 1187.597,A -85,B 0,C 180,E1 28721.666,E2 28721.666} C_VEL
LIN {X 0,Y 608.013,Z 1194.695,A -85,B 0,C 180,E1 28718.988,E2 28718.988} C_VEL
LIN {X 0,Y 607.943,Z 1199.392,A -85,B 0,C 180,E1 28716.611,E2 28716.611} C_VEL
LIN {X 0,Y 607.918,Z 1202.687,A -85,B 0,C 180,E1 28714.245,E2 28714.245} C_VEL
LIN {X 0,Y 607.908,Z 1204.601,A -85,B 0,C 180,E1 28711.697,E2 28711.697} C_VEL
LIN {X 0,Y 607.893,Z 1204.872,A -85,B 0,C 180,E1 28709.435,E2 28709.435} C_VEL
LIN {X 0,Y 607.912,Z 1203.998,A -85,B 0,C 180,E1 28707.266,E2 28707.266} C_VEL
LIN {X 0,Y 607.924,Z 1201.779,A -85,B 0,C 180,E1 28704.999,E2 28704.999} C_VEL
LIN {X 0,Y 607.963,Z 1197.735,A -85,B 0,C 180,E1 28702.44,E2 28702.44} C_VEL
LIN {X 0,Y 608.07,Z 1192.121,A -85,B 0,C 180,E1 28699.962,E2 28699.962} C_VEL
LIN {X 0,Y 608.252,Z 1185.488,A -85,B 0,C 180,E1 28697.661,E2 28697.661} C_VEL
LIN {X 0,Y 608.607,Z 1177.375,A -85,B 0,C 180,E1 28695.345,E2 28695.345} C_VEL
LIN {X 0,Y 609.192,Z 1166.372,A -85,B 0,C 180,E1 28692.718,E2 28692.718} C_VEL
LIN {X 0,Y 609.902,Z 1155.793,A -85,B 0,C 180,E1 28690.562,E2 28690.562} C_VEL
LIN {X 0,Y 610.802,Z 1144.286,A -85,B 0,C 180,E1 28688.489,E2 28688.489} C_VEL
LIN {X 0,Y 612.149,Z 1129.295,A -85,B 0,C 180,E1 28686.104,E2 28686.104} C_VEL
LIN {X 0,Y 613.765,Z 1112.976,A -85,B 0,C 180,E1 28683.85,E2 28683.85} C_VEL
LIN {X 0,Y 615.429,Z 1097.312,A -85,B 0,C 180,E1 28681.911,E2 28681.911} C_VEL
LIN {X 0,Y 617.803,Z 1076.854,A -85,B 0,C 180,E1 28679.673,E2 28679.673} C_VEL
LIN {X 0,Y 619.889,Z 1059.056,A -85,B 0,C 180,E1 28677.95,E2 28677.95} C_VEL
LIN {X 0,Y 621.966,Z 1041.618,A -85,B 0,C 180,E1 28676.427,E2 28676.427} C_VEL
LIN {X 0,Y 624.674,Z 1019.548,A -85,B 0,C 180,E1 28674.703,E2 28674.703} C_VEL
LIN {X 0,Y 627.36,Z 996.425,A -85,B 0,C 180,E1 28673.139,E2 28673.139} C_VEL
LIN {X 0,Y 629.49,Z 977.555,A -85,B 0,C 180,E1 28672.007,E2 28672.007} C_VEL
LIN {X 0,Y 631.514,Z 958.701,A -85,B 0,C 180,E1 28670.998,E2 28670.998} C_VEL
LIN {X 0,Y 633.556,Z 938.34,A -85,B 0,C 180,E1 28670.036,E2 28670.036} C_VEL
LIN {X 0,Y 635.906,Z 913.021,A -85,B 0,C 180,E1 28669.004,E2 28669.004} C_VEL
LIN {X 0,Y 637.949,Z 886.565,A -85,B 0,C 180,E1 28668.131,E2 28668.131} C_VEL
LIN {X 0,Y 639.426,Z 864.549,A -85,B 0,C 180,E1 28667.541,E2 28667.541} C_VEL
LIN {X 0,Y 640.643,Z 842.479,A -85,B 0,C 180,E1 28667.068,E2 28667.068} C_VEL
LIN {X 0,Y 641.744,Z 815.018,A -85,B 0,C 180,E1 28666.629,E2 28666.629} C_VEL
LIN {X 0,Y 645.485,Z 627.653,A -85,B 0,C 180,E1 28664.122,E2 28664.122} C_VEL
LIN {X 0,Y 649.647,Z 417.301,A -85,B 0,C 180,E1 28661.263,E2 28661.263} C_VEL
LIN {X 0,Y 650.124,Z 387.675,A -85,B 0,C 180,E1 28660.839,E2 28660.839} C_VEL
LIN {X 0,Y 645.859,Z 368.248,A -85,B 0,C 180,E1 28660.122,E2 28660.122} C_VEL
LIN {X 0,Y 632.789,Z 349.716,A -85,B 0,C 180,E1 28658.504,E2 28658.504} C_VEL
LIN {X 0,Y 625.129,Z 334.472,A -85,B 0,C 180,E1 28656.514,E2 28656.514} C_VEL
LIN {X 0,Y 615.977,Z 316.986,A -85,B 0,C 180,E1 28654.058,E2 28654.058} C_VEL
LIN {X 0,Y 611.084,Z 307.754,A -85,B 0,C 180,E1 28652.681,E2 28652.681} C_VEL
LIN {X 0,Y 609.196,Z 304.116,A -85,B 0,C 180,E1 28652.124,E2 28652.124} C_VEL
LIN {X 0,Y 609.06,Z 303.412,A -85,B 0,C 180,E1 28651.913,E2 28651.913} C_VEL
LIN {X 0,Y 609.063,Z 303.362,A -85,B 0,C 180,E1 28648.859,E2 28648.859} C_VEL
LIN {X 0,Y 609.054,Z 303.333,A -85,B 0,C 180,E1 28645.675,E2 28645.675} C_VEL
LIN {X 0,Y 609.055,Z 303.326,A -85,B 0,C 180,E1 28642.592,E2 28642.592} C_VEL
LIN {X 0,Y 609.059,Z 303.357,A -85,B 0,C 180,E1 28639.467,E2 28639.467} C_VEL
LIN {X 0,Y 609.055,Z 303.311,A -85,B 0,C 180,E1 28636.304,E2 28636.304} C_VEL
LIN {X 0,Y 609.067,Z 303.36,A -85,B 0,C 180,E1 28633.094,E2 28633.094} C_VEL
LIN {X 0,Y 609.067,Z 303.306,A -85,B 0,C 180,E1 28629.831,E2 28629.831} C_VEL
LIN {X 0,Y 609.064,Z 303.364,A -85,B 0,C 180,E1 28626.599,E2 28626.599} C_VEL
LIN {X 0,Y 609.068,Z 303.357,A -85,B 0,C 180,E1 28623.388,E2 28623.388} C_VEL
LIN {X 0,Y 609.05,Z 303.362,A -85,B 0,C 180,E1 28620.188,E2 28620.188} C_VEL
LIN {X 0,Y 609.066,Z 303.349,A -85,B 0,C 180,E1 28617.054,E2 28617.054} C_VEL
LIN {X 0,Y 609.045,Z 303.352,A -85,B 0,C 180,E1 28613.874,E2 28613.874} C_VEL
LIN {X 0,Y 609.069,Z 303.354,A -85,B 0,C 180,E1 28610.742,E2 28610.742} C_VEL
LIN {X 0,Y 609.046,Z 303.357,A -85,B 0,C 180,E1 28607.58,E2 28607.58} C_VEL
LIN {X 0,Y 609.073,Z 303.36,A -85,B 0,C 180,E1 28604.381,E2 28604.381} C_VEL
LIN {X 0,Y 609.054,Z 303.362,A -85,B 0,C 180,E1 28601.23,E2 28601.23} C_VEL
LIN {X 0,Y 609.051,Z 303.365,A -85,B 0,C 180,E1 28597.917,E2 28597.917} C_VEL
LIN {X 0,Y 609.068,Z 303.308,A -85,B 0,C 180,E1 28594.733,E2 28594.733} C_VEL
LIN {X 0,Y 609.038,Z 303.365,A -85,B 0,C 180,E1 28591.568,E2 28591.568} C_VEL
LIN {X 0,Y 609.073,Z 303.311,A -85,B 0,C 180,E1 28588.53,E2 28588.53} C_VEL
LIN {X 0,Y 609.031,Z 303.364,A -85,B 0,C 180,E1 28585.336,E2 28585.336} C_VEL
LIN {X 0,Y 609.072,Z 303.318,A -85,B 0,C 180,E1 28582.241,E2 28582.241} C_VEL
LIN {X 0,Y 609.024,Z 303.341,A -85,B 0,C 180,E1 28579.186,E2 28579.186} C_VEL
LIN {X 0,Y 609.077,Z 303.353,A -85,B 0,C 180,E1 28576.109,E2 28576.109} C_VEL
LIN {X 0,Y 609.114,Z 303.601,A -85,B 0,C 180,E1 28573.956,E2 28573.956} C_VEL
LIN {X 0,Y 610.635,Z 307.231,A -85,B 0,C 180,E1 28573.362,E2 28573.362} C_VEL
LIN {X 0,Y 615.684,Z 317.194,A -85,B 0,C 180,E1 28571.804,E2 28571.804} C_VEL
LIN {X 0,Y 623.993,Z 334.464,A -85,B 0,C 180,E1 28569.289,E2 28569.289} C_VEL
LIN {X 0,Y 630.161,Z 347.536,A -85,B 0,C 180,E1 28567.532,E2 28567.532} C_VEL
LIN {X 0,Y 630.453,Z 347.987,A -85,B 0,C 180,E1 28567.494,E2 28567.494} C_VEL
LIN {X 0,Y 632.52,Z 352.578,A -85,B 0,C 180,E1 28567.21,E2 28567.21} C_VEL
LIN {X 0,Y 634.377,Z 361.502,A -85,B 0,C 180,E1 28566.879,E2 28566.879} C_VEL
LIN {X 0,Y 635.77,Z 369.283,A -85,B 0,C 180,E1 28566.616,E2 28566.616} C_VEL
LIN {X 0,Y 639.372,Z 386.557,A -85,B 0,C 180,E1 28565.992,E2 28565.992} C_VEL
LIN {X 0,Y 633.816,Z 621.477,A -85,B 0,C 180,E1 28562.806,E2 28562.806} C_VEL
LIN {X 0,Y 630.075,Z 781.855,A -85,B 0,C 180,E1 28560.644,E2 28560.644} C_VEL
LIN {X 0,Y 628.838,Z 808.519,A -85,B 0,C 180,E1 28560.138,E2 28560.138} C_VEL
LIN {X 0,Y 627.363,Z 831.077,A -85,B 0,C 180,E1 28559.555,E2 28559.555} C_VEL
LIN {X 0,Y 625.823,Z 850.976,A -85,B 0,C 180,E1 28558.924,E2 28558.924} C_VEL
LIN {X 0,Y 623.856,Z 873.676,A -85,B 0,C 180,E1 28558.06,E2 28558.06} C_VEL
LIN {X 0,Y 621.48,Z 897.128,A -85,B 0,C 180,E1 28556.981,E2 28556.981} C_VEL
LIN {X 0,Y 619.44,Z 915.618,A -85,B 0,C 180,E1 28555.991,E2 28555.991} C_VEL
LIN {X 0,Y 617.342,Z 933.565,A -85,B 0,C 180,E1 28554.903,E2 28554.903} C_VEL
LIN {X 0,Y 614.527,Z 957.787,A -85,B 0,C 180,E1 28553.245,E2 28553.245} C_VEL
LIN {X 0,Y 612.313,Z 976.769,A -85,B 0,C 180,E1 28551.757,E2 28551.757} C_VEL
LIN {X 0,Y 610.324,Z 994.226,A -85,B 0,C 180,E1 28550.223,E2 28550.223} C_VEL
LIN {X 0,Y 608.02,Z 1014.398,A -85,B 0,C 180,E1 28548.207,E2 28548.207} C_VEL
LIN {X 0,Y 606.333,Z 1029.668,A -85,B 0,C 180,E1 28546.477,E2 28546.477} C_VEL
LIN {X 0,Y 604.652,Z 1046.31,A -85,B 0,C 180,E1 28544.362,E2 28544.362} C_VEL
LIN {X 0,Y 603.273,Z 1060.722,A -85,B 0,C 180,E1 28542.248,E2 28542.248} C_VEL
LIN {X 0,Y 602.289,Z 1072.346,A -85,B 0,C 180,E1 28540.328,E2 28540.328} C_VEL
LIN {X 0,Y 601.368,Z 1085.02,A -85,B 0,C 180,E1 28537.932,E2 28537.932} C_VEL
LIN {X 0,Y 600.785,Z 1094.881,A -85,B 0,C 180,E1 28535.731,E2 28535.731} C_VEL
LIN {X 0,Y 600.391,Z 1102.959,A -85,B 0,C 180,E1 28533.628,E2 28533.628} C_VEL
LIN {X 0,Y 600.117,Z 1110.819,A -85,B 0,C 180,E1 28531.146,E2 28531.146} C_VEL
LIN {X 0,Y 599.993,Z 1116.233,A -85,B 0,C 180,E1 28528.95,E2 28528.95} C_VEL
LIN {X 0,Y 599.932,Z 1120.054,A -85,B 0,C 180,E1 28526.943,E2 28526.943} C_VEL
LIN {X 0,Y 599.91,Z 1123.014,A -85,B 0,C 180,E1 28524.74,E2 28524.74} C_VEL
LIN {X 0,Y 599.912,Z 1124.703,A -85,B 0,C 180,E1 28522.241,E2 28522.241} C_VEL
LIN {X 0,Y 599.893,Z 1124.832,A -85,B 0,C 180,E1 28520.212,E2 28520.212} C_VEL
LIN {X 0,Y 599.91,Z 1123.861,A -85,B 0,C 180,E1 28518.17,E2 28518.17} C_VEL
LIN {X 0,Y 599.915,Z 1121.53,A -85,B 0,C 180,E1 28515.917,E2 28515.917} C_VEL
LIN {X 0,Y 599.98,Z 1117.151,A -85,B 0,C 180,E1 28513.389,E2 28513.389} C_VEL
LIN {X 0,Y 600.081,Z 1112.339,A -85,B 0,C 180,E1 28511.342,E2 28511.342} C_VEL
LIN {X 0,Y 600.25,Z 1106.449,A -85,B 0,C 180,E1 28509.321,E2 28509.321} C_VEL
LIN {X 0,Y 600.641,Z 1097.728,A -85,B 0,C 180,E1 28506.868,E2 28506.868} C_VEL
LIN {X 0,Y 601.167,Z 1088.364,A -85,B 0,C 180,E1 28504.695,E2 28504.695} C_VEL
LIN {X 0,Y 601.817,Z 1078.523,A -85,B 0,C 180,E1 28502.707,E2 28502.707} C_VEL
LIN {X 0,Y 602.888,Z 1065.31,A -85,B 0,C 180,E1 28500.382,E2 28500.382} C_VEL
LIN {X 0,Y 604.122,Z 1051.529,A -85,B 0,C 180,E1 28498.291,E2 28498.291} C_VEL
LIN {X 0,Y 605.516,Z 1037.646,A -85,B 0,C 180,E1 28496.415,E2 28496.415} C_VEL
LIN {X 0,Y 607.51,Z 1018.928,A -85,B 0,C 180,E1 28494.196,E2 28494.196} C_VEL
LIN {X 0,Y 609.272,Z 1003.213,A -85,B 0,C 180,E1 28492.554,E2 28492.554} C_VEL
LIN {X 0,Y 611.466,Z 984.609,A -85,B 0,C 180,E1 28490.815,E2 28490.815} C_VEL
LIN {X 0,Y 613.782,Z 964.237,A -85,B 0,C 180,E1 28489.152,E2 28489.152} C_VEL
LIN {X 0,Y 616.149,Z 943.65,A -85,B 0,C 180,E1 28487.667,E2 28487.667} C_VEL
LIN {X 0,Y 619.032,Z 919.563,A -85,B 0,C 180,E1 28486.138,E2 28486.138} C_VEL
LIN {X 0,Y 621.17,Z 900.541,A -85,B 0,C 180,E1 28485.094,E2 28485.094} C_VEL
LIN {X 0,Y 623.174,Z 881.414,A -85,B 0,C 180,E1 28484.177,E2 28484.177} C_VEL
LIN {X 0,Y 625.526,Z 856.577,A -85,B 0,C 180,E1 28483.169,E2 28483.169} C_VEL
LIN {X 0,Y 627.283,Z 834.158,A -85,B 0,C 180,E1 28482.431,E2 28482.431} C_VEL
LIN {X 0,Y 628.587,Z 814.804,A -85,B 0,C 180,E1 28481.909,E2 28481.909} C_VEL
LIN {X 0,Y 629.703,Z 794.519,A -85,B 0,C 180,E1 28481.471,E2 28481.471} C_VEL
LIN {X 0,Y 630.747,Z 765.624,A -85,B 0,C 180,E1 28481.015,E2 28481.015} C_VEL
LIN {X 0,Y 636.371,Z 524.604,A -85,B 0,C 180,E1 28477.77,E2 28477.77} C_VEL
LIN {X 0,Y 639.791,Z 385.356,A -85,B 0,C 180,E1 28475.844,E2 28475.844} C_VEL
LIN {X 0,Y 635.875,Z 367.334,A -85,B 0,C 180,E1 28475.136,E2 28475.136} C_VEL
LIN {X 0,Y 625.687,Z 352.026,A -85,B 0,C 180,E1 28473.734,E2 28473.734} C_VEL
LIN {X 0,Y 622.334,Z 347.044,A -85,B 0,C 180,E1 28473.222,E2 28473.222} C_VEL
LIN {X 0,Y 616.44,Z 334.56,A -85,B 0,C 180,E1 28471.264,E2 28471.264} C_VEL
LIN {X 0,Y 610.872,Z 323.175,A -85,B 0,C 180,E1 28469.302,E2 28469.302} C_VEL
LIN {X 0,Y 607.631,Z 317.343,A -85,B 0,C 180,E1 28468.182,E2 28468.182} C_VEL
LIN {X 0,Y 605.938,Z 313.804,A -85,B 0,C 180,E1 28467.519,E2 28467.519} C_VEL
LIN {X 0,Y 603.925,Z 310.084,A -85,B 0,C 180,E1 28466.766,E2 28466.766} C_VEL
LIN {X 0,Y 601.287,Z 305.213,A -85,B 0,C 180,E1 28465.723,E2 28465.723} C_VEL
LIN {X 0,Y 601.146,Z 304.48,A -85,B 0,C 180,E1 28465.518,E2 28465.518} C_VEL
LIN {X 0,Y 601.12,Z 304.315,A -85,B 0,C 180,E1 28462.287,E2 28462.287} C_VEL
LIN {X 0,Y 601.134,Z 304.351,A -85,B 0,C 180,E1 28459.027,E2 28459.027} C_VEL
LIN {X 0,Y 601.127,Z 304.324,A -85,B 0,C 180,E1 28455.731,E2 28455.731} C_VEL
LIN {X 0,Y 601.115,Z 304.311,A -85,B 0,C 180,E1 28452.488,E2 28452.488} C_VEL
LIN {X 0,Y 601.122,Z 304.352,A -85,B 0,C 180,E1 28449.285,E2 28449.285} C_VEL
LIN {X 0,Y 601.113,Z 304.312,A -85,B 0,C 180,E1 28446.111,E2 28446.111} C_VEL
LIN {X 0,Y 601.12,Z 304.331,A -85,B 0,C 180,E1 28442.956,E2 28442.956} C_VEL
LIN {X 0,Y 601.126,Z 304.338,A -85,B 0,C 180,E1 28439.714,E2 28439.714} C_VEL
LIN {X 0,Y 601.127,Z 304.306,A -85,B 0,C 180,E1 28436.472,E2 28436.472} C_VEL
LIN {X 0,Y 601.127,Z 304.352,A -85,B 0,C 180,E1 28433.122,E2 28433.122} C_VEL
LIN {X 0,Y 601.122,Z 304.31,A -85,B 0,C 180,E1 28429.941,E2 28429.941} C_VEL
LIN {X 0,Y 601.117,Z 304.334,A -85,B 0,C 180,E1 28426.827,E2 28426.827} C_VEL
LIN {X 0,Y 601.125,Z 304.339,A -85,B 0,C 180,E1 28423.674,E2 28423.674} C_VEL
LIN {X 0,Y 601.11,Z 304.309,A -85,B 0,C 180,E1 28420.568,E2 28420.568} C_VEL
LIN {X 0,Y 601.126,Z 304.343,A -85,B 0,C 180,E1 28417.389,E2 28417.389} C_VEL
LIN {X 0,Y 601.116,Z 304.332,A -85,B 0,C 180,E1 28414.163,E2 28414.163} C_VEL
LIN {X 0,Y 601.13,Z 304.31,A -85,B 0,C 180,E1 28410.942,E2 28410.942} C_VEL
LIN {X 0,Y 601.172,Z 304.686,A -85,B 0,C 180,E1 28409.925,E2 28409.925} C_VEL
LIN {X 0,Y 602.699,Z 308.21,A -85,B 0,C 180,E1 28409.243,E2 28409.243} C_VEL
LIN {X 0,Y 604.13,Z 310.212,A -85,B 0,C 180,E1 28408.799,E2 28408.799} C_VEL
LIN {X 0,Y 606.016,Z 313.786,A -85,B 0,C 180,E1 28408.131,E2 28408.131} C_VEL
LIN {X 0,Y 607.16,Z 315.769,A -85,B 0,C 180,E1 28407.753,E2 28407.753} C_VEL
LIN {X 0,Y 610.022,Z 321.047,A -85,B 0,C 180,E1 28406.807,E2 28406.807} C_VEL
LIN {X 0,Y 614.573,Z 329.233,A -85,B 0,C 180,E1 28405.402,E2 28405.402} C_VEL
LIN {X 0,Y 621.037,Z 342.066,A -85,B 0,C 180,E1 28403.436,E2 28403.436} C_VEL
LIN {X 0,Y 625.139,Z 350.363,A -85,B 0,C 180,E1 28402.309,E2 28402.309} C_VEL
LIN {X 0,Y 641.047,Z 373.558,A -85,B 0,C 180,E1 28400.223,E2 28400.223} C_VEL
LIN {X 0,Y 644.537,Z 391.105,A -85,B 0,C 180,E1 28399.604,E2 28399.604} C_VEL
LIN {X 0,Y 640.048,Z 603.695,A -85,B 0,C 180,E1 28396.687,E2 28396.687} C_VEL
LIN {X 0,Y 635.8,Z 818.716,A -85,B 0,C 180,E1 28393.813,E2 28393.813} C_VEL
